LIN {X 0,Y 574.042,Z 450.55,A -85,B 0,C 180,E1 -1993.505,E2 -1993.505} C_VEL
LIN {X 0,Y 573.917,Z 424.53,A -85,B 0,C 180,E1 -1993.836,E2 -1993.836} C_VEL
LIN {X 0,Y 573.507,Z 421.165,A -85,B 0,C 180,E1 -1993.916,E2 -1993.916} C_VEL
LIN {X 0,Y 573.675,Z 396.566,A -85,B 0,C 180,E1 -1996.915,E2 -1996.915} C_VEL
LIN {X 0,Y 573.955,Z 372.952,A -85,B 0,C 180,E1 -1999.849,E2 -1999.849} C_VEL
LIN {X 0,Y 574.301,Z 350.569,A -85,B 0,C 180,E1 -2002.674,E2 -2002.674} C_VEL
LIN {X 0,Y 574.39,Z 334.005,A -85,B 0,C 180,E1 -2004.75,E2 -2004.75} C_VEL
LIN {X 0,Y 573.247,Z 327.79,A -85,B 0,C 180,E1 -2005.605,E2 -2005.605} C_VEL
LIN {X 0,Y 573.252,Z 327.703,A -85,B 0,C 180,E1 -2008.028,E2 -2008.028} C_VEL
LIN {X 0,Y 573.25,Z 327.705,A -85,B 0,C 180,E1 -2010.176,E2 -2010.176} C_VEL
LIN {X 0,Y 573.259,Z 327.704,A -85,B 0,C 180,E1 -2012.645,E2 -2012.645} C_VEL
LIN {X 0,Y 573.21,Z 327.704,A -85,B 0,C 180,E1 -2015.188,E2 -2015.188} C_VEL
LIN {X 0,Y 573.239,Z 327.702,A -85,B 0,C 180,E1 -2017.807,E2 -2017.807} C_VEL
LIN {X 0,Y 573.25,Z 327.704,A -85,B 0,C 180,E1 -2020.525,E2 -2020.525} C_VEL
LIN {X 0,Y 573.245,Z 327.698,A -85,B 0,C 180,E1 -2023.359,E2 -2023.359} C_VEL
LIN {X 0,Y 573.243,Z 327.706,A -85,B 0,C 180,E1 -2026.331,E2 -2026.331} C_VEL
LIN {X 0,Y 573.233,Z 327.703,A -85,B 0,C 180,E1 -2028.542,E2 -2028.542} C_VEL
LIN {X 0,Y 573.248,Z 327.698,A -85,B 0,C 180,E1 -2031.298,E2 -2031.298} C_VEL
LIN {X 0,Y 573.245,Z 327.707,A -85,B 0,C 180,E1 -2034.014,E2 -2034.014} C_VEL
LIN {X 0,Y 573.275,Z 327.697,A -85,B 0,C 180,E1 -2036.517,E2 -2036.517} C_VEL
LIN {X 0,Y 573.234,Z 327.701,A -85,B 0,C 180,E1 -2039.117,E2 -2039.117} C_VEL
LIN {X 0,Y 573.242,Z 327.697,A -85,B 0,C 180,E1 -2041.435,E2 -2041.435} C_VEL
LIN {X 0,Y 573.269,Z 327.702,A -85,B 0,C 180,E1 -2043.81,E2 -2043.81} C_VEL
LIN {X 0,Y 573.238,Z 327.706,A -85,B 0,C 180,E1 -2046.134,E2 -2046.134} C_VEL
LIN {X 0,Y 573.29,Z 327.923,A -85,B 0,C 180,E1 -2046.936,E2 -2046.936} C_VEL
LIN {X 0,Y 574.042,Z 332.774,A -85,B 0,C 180,E1 -2047.694,E2 -2047.694} C_VEL
LIN {X 0,Y 573.791,Z 353.69,A -85,B 0,C 180,E1 -2050.688,E2 -2050.688} C_VEL
LIN {X 0,Y 573.581,Z 371.938,A -85,B 0,C 180,E1 -2053.24,E2 -2053.24} C_VEL
LIN {X 0,Y 573.876,Z 374.016,A -85,B 0,C 180,E1 -2053.322,E2 -2053.322} C_VEL
LIN {X 0,Y 574.602,Z 377.936,A -85,B 0,C 180,E1 -2053.393,E2 -2053.393} C_VEL
LIN {X 0,Y 574.275,Z 508.286,A -85,B 0,C 180,E1 -2055.062,E2 -2055.062} C_VEL
LIN {X 0,Y 574.177,Z 521.251,A -85,B 0,C 180,E1 -2055.339,E2 -2055.339} C_VEL
LIN {X 0,Y 574.097,Z 535.103,A -85,B 0,C 180,E1 -2055.771,E2 -2055.771} C_VEL
LIN {X 0,Y 573.926,Z 548.919,A -85,B 0,C 180,E1 -2056.365,E2 -2056.365} C_VEL
LIN {X 0,Y 573.742,Z 560.44,A -85,B 0,C 180,E1 -2056.991,E2 -2056.991} C_VEL
LIN {X 0,Y 573.599,Z 571.257,A -85,B 0,C 180,E1 -2057.708,E2 -2057.708} C_VEL
LIN {X 0,Y 573.455,Z 581.621,A -85,B 0,C 180,E1 -2058.53,E2 -2058.53} C_VEL
LIN {X 0,Y 573.355,Z 590.92,A -85,B 0,C 180,E1 -2059.404,E2 -2059.404} C_VEL
LIN {X 0,Y 573.256,Z 600.453,A -85,B 0,C 180,E1 -2060.472,E2 -2060.472} C_VEL
LIN {X 0,Y 573.143,Z 609.469,A -85,B 0,C 180,E1 -2061.715,E2 -2061.715} C_VEL
LIN {X 0,Y 573.091,Z 614.888,A -85,B 0,C 180,E1 -2062.601,E2 -2062.601} C_VEL
LIN {X 0,Y 573.022,Z 620.311,A -85,B 0,C 180,E1 -2063.662,E2 -2063.662} C_VEL
LIN {X 0,Y 573,Z 624.764,A -85,B 0,C 180,E1 -2064.721,E2 -2064.721} C_VEL
LIN {X 0,Y 573.029,Z 628.315,A -85,B 0,C 180,E1 -2065.779,E2 -2065.779} C_VEL
LIN {X 0,Y 572.957,Z 631.716,A -85,B 0,C 180,E1 -2067.187,E2 -2067.187} C_VEL
LIN {X 0,Y 572.939,Z 632.942,A -85,B 0,C 180,E1 -2067.89,E2 -2067.89} C_VEL
LIN {X 0,Y 572.936,Z 634.281,A -85,B 0,C 180,E1 -2069.296,E2 -2069.296} C_VEL
LIN {X 0,Y 572.937,Z 634.496,A -85,B 0,C 180,E1 -2069.999,E2 -2069.999} C_VEL
LIN {X 0,Y 572.941,Z 633.863,A -85,B 0,C 180,E1 -2071.405,E2 -2071.405} C_VEL
LIN {X 0,Y 572.954,Z 631.893,A -85,B 0,C 180,E1 -2072.811,E2 -2072.811} C_VEL
LIN {X 0,Y 573.008,Z 630.437,A -85,B 0,C 180,E1 -2073.515,E2 -2073.515} C_VEL
LIN {X 0,Y 572.955,Z 626.342,A -85,B 0,C 180,E1 -2074.925,E2 -2074.925} C_VEL
LIN {X 0,Y 573.044,Z 622.298,A -85,B 0,C 180,E1 -2075.983,E2 -2075.983} C_VEL
LIN {X 0,Y 573.053,Z 617.286,A -85,B 0,C 180,E1 -2077.044,E2 -2077.044} C_VEL
LIN {X 0,Y 573.128,Z 611.185,A -85,B 0,C 180,E1 -2078.106,E2 -2078.106} C_VEL
LIN {X 0,Y 573.219,Z 603.876,A -85,B 0,C 180,E1 -2079.17,E2 -2079.17} C_VEL
LIN {X 0,Y 573.303,Z 595.124,A -85,B 0,C 180,E1 -2080.238,E2 -2080.238} C_VEL
LIN {X 0,Y 573.487,Z 583.882,A -85,B 0,C 180,E1 -2081.365,E2 -2081.365} C_VEL
LIN {X 0,Y 573.585,Z 572.521,A -85,B 0,C 180,E1 -2082.291,E2 -2082.291} C_VEL
LIN {X 0,Y 573.735,Z 561.93,A -85,B 0,C 180,E1 -2083.007,E2 -2083.007} C_VEL
LIN {X 0,Y 573.88,Z 550.7,A -85,B 0,C 180,E1 -2083.634,E2 -2083.634} C_VEL
LIN {X 0,Y 574.013,Z 538.844,A -85,B 0,C 180,E1 -2084.173,E2 -2084.173} C_VEL
LIN {X 0,Y 574.186,Z 523.882,A -85,B 0,C 180,E1 -2084.684,E2 -2084.684} C_VEL
LIN {X 0,Y 574.28,Z 509.711,A -85,B 0,C 180,E1 -2085.004,E2 -2085.004} C_VEL
LIN {X 0,Y 574.423,Z 457.939,A -85,B 0,C 180,E1 -2085.682,E2 -2085.682} C_VEL
LIN {X 0,Y 574.434,Z 376.847,A -85,B 0,C 180,E1 -2086.716,E2 -2086.716} C_VEL
LIN {X 0,Y 573.637,Z 372.312,A -85,B 0,C 180,E1 -2086.819,E2 -2086.819} C_VEL
LIN {X 0,Y 573.702,Z 359.568,A -85,B 0,C 180,E1 -2088.572,E2 -2088.572} C_VEL
LIN {X 0,Y 573.962,Z 340.021,A -85,B 0,C 180,E1 -2091.352,E2 -2091.352} C_VEL
LIN {X 0,Y 574.053,Z 332.1,A -85,B 0,C 180,E1 -2092.493,E2 -2092.493} C_VEL
LIN {X 0,Y 573.275,Z 327.837,A -85,B 0,C 180,E1 -2093.182,E2 -2093.182} C_VEL
LIN {X 0,Y 573.255,Z 327.7,A -85,B 0,C 180,E1 -2095.409,E2 -2095.409} C_VEL
LIN {X 0,Y 573.263,Z 327.705,A -85,B 0,C 180,E1 -2098.031,E2 -2098.031} C_VEL
LIN {X 0,Y 573.243,Z 327.7,A -85,B 0,C 180,E1 -2100.884,E2 -2100.884} C_VEL
LIN {X 0,Y 573.285,Z 327.695,A -85,B 0,C 180,E1 -2103.527,E2 -2103.527} C_VEL
LIN {X 0,Y 573.258,Z 327.705,A -85,B 0,C 180,E1 -2106.047,E2 -2106.047} C_VEL
LIN {X 0,Y 573.246,Z 327.699,A -85,B 0,C 180,E1 -2108.7,E2 -2108.7} C_VEL
LIN {X 0,Y 573.249,Z 327.702,A -85,B 0,C 180,E1 -2111.595,E2 -2111.595} C_VEL
LIN {X 0,Y 573.233,Z 327.7,A -85,B 0,C 180,E1 -2114.332,E2 -2114.332} C_VEL
LIN {X 0,Y 573.254,Z 327.699,A -85,B 0,C 180,E1 -2117.355,E2 -2117.355} C_VEL
LIN {X 0,Y 573.243,Z 327.698,A -85,B 0,C 180,E1 -2120.392,E2 -2120.392} C_VEL
LIN {X 0,Y 573.249,Z 327.695,A -85,B 0,C 180,E1 -2123.077,E2 -2123.077} C_VEL
LIN {X 0,Y 573.265,Z 327.706,A -85,B 0,C 180,E1 -2125.671,E2 -2125.671} C_VEL
LIN {X 0,Y 573.244,Z 327.699,A -85,B 0,C 180,E1 -2128.185,E2 -2128.185} C_VEL
LIN {X 0,Y 573.262,Z 327.69,A -85,B 0,C 180,E1 -2130.634,E2 -2130.634} C_VEL
LIN {X 0,Y 573.264,Z 327.702,A -85,B 0,C 180,E1 -2133.499,E2 -2133.499} C_VEL
LIN {X 0,Y 573.236,Z 327.701,A -85,B 0,C 180,E1 -2136.135,E2 -2136.135} C_VEL
LIN {X 0,Y 573.251,Z 327.697,A -85,B 0,C 180,E1 -2138.706,E2 -2138.706} C_VEL
LIN {X 0,Y 573.233,Z 327.71,A -85,B 0,C 180,E1 -2141.411,E2 -2141.411} C_VEL
LIN {X 0,Y 573.252,Z 327.701,A -85,B 0,C 180,E1 -2143.622,E2 -2143.622} C_VEL
LIN {X 0,Y 573.231,Z 327.7,A -85,B 0,C 180,E1 -2146.529,E2 -2146.529} C_VEL
LIN {X 0,Y 573.272,Z 327.7,A -85,B 0,C 180,E1 -2149.403,E2 -2149.403} C_VEL
LIN {X 0,Y 573.282,Z 327.693,A -85,B 0,C 180,E1 -2152.25,E2 -2152.25} C_VEL
LIN {X 0,Y 573.307,Z 327.7,A -85,B 0,C 180,E1 -2155.077,E2 -2155.077} C_VEL
LIN {X 0,Y 573.301,Z 327.691,A -85,B 0,C 180,E1 -2157.892,E2 -2157.892} C_VEL
LIN {X 0,Y 573.333,Z 327.693,A -85,B 0,C 180,E1 -2160.702,E2 -2160.702} C_VEL
LIN {X 0,Y 573.237,Z 327.7,A -85,B 0,C 180,E1 -2163.514,E2 -2163.514} C_VEL
LIN {X 0,Y 573.288,Z 327.694,A -85,B 0,C 180,E1 -2165.628,E2 -2165.628} C_VEL
LIN {X 0,Y 573.299,Z 327.695,A -85,B 0,C 180,E1 -2168.459,E2 -2168.459} C_VEL
LIN {X 0,Y 573.288,Z 327.695,A -85,B 0,C 180,E1 -2171.312,E2 -2171.312} C_VEL
LIN {X 0,Y 573.271,Z 327.699,A -85,B 0,C 180,E1 -2174.425,E2 -2174.425} C_VEL
LIN {X 0,Y 573.252,Z 327.701,A -85,B 0,C 180,E1 -2177.112,E2 -2177.112} C_VEL
LIN {X 0,Y 573.25,Z 327.699,A -85,B 0,C 180,E1 -2180.077,E2 -2180.077} C_VEL
LIN {X 0,Y 573.262,Z 327.698,A -85,B 0,C 180,E1 -2183.154,E2 -2183.154} C_VEL
LIN {X 0,Y 573.28,Z 327.698,A -85,B 0,C 180,E1 -2186.189,E2 -2186.189} C_VEL
LIN {X 0,Y 573.235,Z 327.701,A -85,B 0,C 180,E1 -2188.565,E2 -2188.565} C_VEL
LIN {X 0,Y 573.229,Z 327.701,A -85,B 0,C 180,E1 -2190.993,E2 -2190.993} C_VEL
LIN {X 0,Y 573.279,Z 327.695,A -85,B 0,C 180,E1 -2193.529,E2 -2193.529} C_VEL
LIN {X 0,Y 573.252,Z 327.702,A -85,B 0,C 180,E1 -2196.049,E2 -2196.049} C_VEL
LIN {X 0,Y 573.241,Z 327.701,A -85,B 0,C 180,E1 -2198.702,E2 -2198.702} C_VEL
LIN {X 0,Y 573.258,Z 327.699,A -85,B 0,C 180,E1 -2201.598,E2 -2201.598} C_VEL
LIN {X 0,Y 573.232,Z 327.704,A -85,B 0,C 180,E1 -2204.334,E2 -2204.334} C_VEL
LIN {X 0,Y 573.237,Z 327.7,A -85,B 0,C 180,E1 -2207.359,E2 -2207.359} C_VEL
LIN {X 0,Y 573.245,Z 327.703,A -85,B 0,C 180,E1 -2210.394,E2 -2210.394} C_VEL
LIN {X 0,Y 573.252,Z 327.698,A -85,B 0,C 180,E1 -2213.079,E2 -2213.079} C_VEL
LIN {X 0,Y 573.272,Z 327.701,A -85,B 0,C 180,E1 -2215.673,E2 -2215.673} C_VEL
LIN {X 0,Y 573.247,Z 327.705,A -85,B 0,C 180,E1 -2218.186,E2 -2218.186} C_VEL
LIN {X 0,Y 573.268,Z 327.691,A -85,B 0,C 180,E1 -2220.636,E2 -2220.636} C_VEL
LIN {X 0,Y 573.267,Z 327.702,A -85,B 0,C 180,E1 -2223.502,E2 -2223.502} C_VEL
LIN {X 0,Y 573.232,Z 327.707,A -85,B 0,C 180,E1 -2226.136,E2 -2226.136} C_VEL
LIN {X 0,Y 573.26,Z 327.868,A -85,B 0,C 180,E1 -2226.875,E2 -2226.875} C_VEL
LIN {X 0,Y 574.085,Z 333.097,A -85,B 0,C 180,E1 -2227.698,E2 -2227.698} C_VEL
LIN {X 0,Y 573.784,Z 354.019,A -85,B 0,C 180,E1 -2230.689,E2 -2230.689} C_VEL
LIN {X 0,Y 573.608,Z 372.016,A -85,B 0,C 180,E1 -2233.203,E2 -2233.203} C_VEL
LIN {X 0,Y 574.046,Z 374.736,A -85,B 0,C 180,E1 -2233.291,E2 -2233.291} C_VEL
LIN {X 0,Y 574.6,Z 379.508,A -85,B 0,C 180,E1 -2233.368,E2 -2233.368} C_VEL
LIN {X 0,Y 574.303,Z 508.7,A -85,B 0,C 180,E1 -2235.019,E2 -2235.019} C_VEL
LIN {X 0,Y 574.186,Z 523.423,A -85,B 0,C 180,E1 -2235.349,E2 -2235.349} C_VEL
LIN {X 0,Y 574.02,Z 537.729,A -85,B 0,C 180,E1 -2235.827,E2 -2235.827} C_VEL
LIN {X 0,Y 573.889,Z 551.665,A -85,B 0,C 180,E1 -2236.456,E2 -2236.456} C_VEL
LIN {X 0,Y 573.717,Z 564.118,A -85,B 0,C 180,E1 -2237.173,E2 -2237.173} C_VEL
LIN {X 0,Y 573.532,Z 576.655,A -85,B 0,C 180,E1 -2238.067,E2 -2238.067} C_VEL
LIN {X 0,Y 573.435,Z 588.186,A -85,B 0,C 180,E1 -2239.084,E2 -2239.084} C_VEL
LIN {X 0,Y 573.239,Z 597.86,A -85,B 0,C 180,E1 -2240.118,E2 -2240.118} C_VEL
LIN {X 0,Y 573.201,Z 606.179,A -85,B 0,C 180,E1 -2241.185,E2 -2241.185} C_VEL
LIN {X 0,Y 573.109,Z 614.133,A -85,B 0,C 180,E1 -2242.426,E2 -2242.426} C_VEL
LIN {X 0,Y 573.02,Z 620.531,A -85,B 0,C 180,E1 -2243.664,E2 -2243.664} C_VEL
LIN {X 0,Y 573.001,Z 624.964,A -85,B 0,C 180,E1 -2244.723,E2 -2244.723} C_VEL
LIN {X 0,Y 573.028,Z 628.447,A -85,B 0,C 180,E1 -2245.781,E2 -2245.781} C_VEL
LIN {X 0,Y 572.956,Z 631.835,A -85,B 0,C 180,E1 -2247.189,E2 -2247.189} C_VEL
LIN {X 0,Y 572.941,Z 633.834,A -85,B 0,C 180,E1 -2248.595,E2 -2248.595} C_VEL
LIN {X 0,Y 572.937,Z 634.5,A -85,B 0,C 180,E1 -2250.001,E2 -2250.001} C_VEL
LIN {X 0,Y 572.941,Z 633.832,A -85,B 0,C 180,E1 -2251.407,E2 -2251.407} C_VEL
LIN {X 0,Y 572.956,Z 631.83,A -85,B 0,C 180,E1 -2252.813,E2 -2252.813} C_VEL
LIN {X 0,Y 573.028,Z 628.44,A -85,B 0,C 180,E1 -2254.221,E2 -2254.221} C_VEL
LIN {X 0,Y 573.059,Z 623.565,A -85,B 0,C 180,E1 -2255.631,E2 -2255.631} C_VEL
LIN {X 0,Y 573.059,Z 618.85,A -85,B 0,C 180,E1 -2256.693,E2 -2256.693} C_VEL
LIN {X 0,Y 573.126,Z 612.031,A -85,B 0,C 180,E1 -2257.93,E2 -2257.93} C_VEL
LIN {X 0,Y 573.226,Z 603.552,A -85,B 0,C 180,E1 -2259.172,E2 -2259.172} C_VEL
LIN {X 0,Y 573.305,Z 594.7,A -85,B 0,C 180,E1 -2260.24,E2 -2260.24} C_VEL
LIN {X 0,Y 573.464,Z 583.982,A -85,B 0,C 180,E1 -2261.309,E2 -2261.309} C_VEL
LIN {X 0,Y 573.618,Z 573.131,A -85,B 0,C 180,E1 -2262.202,E2 -2262.202} C_VEL
LIN {X 0,Y 573.741,Z 561.243,A -85,B 0,C 180,E1 -2263.009,E2 -2263.009} C_VEL
LIN {X 0,Y 573.947,Z 548.081,A -85,B 0,C 180,E1 -2263.725,E2 -2263.725} C_VEL
LIN {X 0,Y 574.085,Z 534.8,A -85,B 0,C 180,E1 -2264.285,E2 -2264.285} C_VEL
LIN {X 0,Y 574.208,Z 520.713,A -85,B 0,C 180,E1 -2264.722,E2 -2264.722} C_VEL
LIN {X 0,Y 574.315,Z 507.08,A -85,B 0,C 180,E1 -2265.005,E2 -2265.005} C_VEL
LIN {X 0,Y 574.467,Z 376.987,A -85,B 0,C 180,E1 -2266.668,E2 -2266.668} C_VEL
LIN {X 0,Y 573.617,Z 372.383,A -85,B 0,C 180,E1 -2266.77,E2 -2266.77} C_VEL
LIN {X 0,Y 573.621,Z 368.522,A -85,B 0,C 180,E1 -2267.266,E2 -2267.266} C_VEL
LIN {X 0,Y 573.892,Z 346.16,A -85,B 0,C 180,E1 -2270.428,E2 -2270.428} C_VEL
LIN {X 0,Y 574.034,Z 331.776,A -85,B 0,C 180,E1 -2272.496,E2 -2272.496} C_VEL
LIN {X 0,Y 573.262,Z 327.809,A -85,B 0,C 180,E1 -2273.15,E2 -2273.15} C_VEL
LIN {X 0,Y 573.258,Z 327.699,A -85,B 0,C 180,E1 -2275.411,E2 -2275.411} C_VEL
LIN {X 0,Y 573.269,Z 327.703,A -85,B 0,C 180,E1 -2278.032,E2 -2278.032} C_VEL
LIN {X 0,Y 573.234,Z 327.701,A -85,B 0,C 180,E1 -2280.883,E2 -2280.883} C_VEL
LIN {X 0,Y 573.267,Z 327.698,A -85,B 0,C 180,E1 -2283.524,E2 -2283.524} C_VEL
LIN {X 0,Y 573.266,Z 327.705,A -85,B 0,C 180,E1 -2286.048,E2 -2286.048} C_VEL
LIN {X 0,Y 573.247,Z 327.7,A -85,B 0,C 180,E1 -2288.702,E2 -2288.702} C_VEL
LIN {X 0,Y 573.234,Z 327.705,A -85,B 0,C 180,E1 -2291.593,E2 -2291.593} C_VEL
LIN {X 0,Y 573.233,Z 327.704,A -85,B 0,C 180,E1 -2294.334,E2 -2294.334} C_VEL
LIN {X 0,Y 573.245,Z 327.702,A -85,B 0,C 180,E1 -2297.359,E2 -2297.359} C_VEL
LIN {X 0,Y 573.243,Z 327.701,A -85,B 0,C 180,E1 -2300.393,E2 -2300.393} C_VEL
LIN {X 0,Y 573.256,Z 327.699,A -85,B 0,C 180,E1 -2303.078,E2 -2303.078} C_VEL
LIN {X 0,Y 573.27,Z 327.706,A -85,B 0,C 180,E1 -2305.671,E2 -2305.671} C_VEL
LIN {X 0,Y 573.245,Z 327.702,A -85,B 0,C 180,E1 -2308.185,E2 -2308.185} C_VEL
LIN {X 0,Y 573.268,Z 327.697,A -85,B 0,C 180,E1 -2310.634,E2 -2310.634} C_VEL
LIN {X 0,Y 573.255,Z 327.702,A -85,B 0,C 180,E1 -2313.024,E2 -2313.024} C_VEL
LIN {X 0,Y 573.3,Z 327.912,A -85,B 0,C 180,E1 -2314.607,E2 -2314.607} C_VEL
LIN {X 0,Y 574.331,Z 334.315,A -85,B 0,C 180,E1 -2315.414,E2 -2315.414} C_VEL
LIN {X 0,Y 574.197,Z 352.833,A -85,B 0,C 180,E1 -2317.702,E2 -2317.702} C_VEL
LIN {X 0,Y 573.943,Z 373.525,A -85,B 0,C 180,E1 -2320.313,E2 -2320.313} C_VEL
LIN {X 0,Y 573.687,Z 397.322,A -85,B 0,C 180,E1 -2323.268,E2 -2323.268} C_VEL
LIN {X 0,Y 573.472,Z 420.909,A -85,B 0,C 180,E1 -2326.151,E2 -2326.151} C_VEL
LIN {X 0,Y 573.649,Z 422.658,A -85,B 0,C 180,E1 -2326.223,E2 -2326.223} C_VEL
LIN {X 0,Y 574.082,Z 429.808,A -85,B 0,C 180,E1 -2326.324,E2 -2326.324} C_VEL
LIN {X 0,Y 573.866,Z 530.384,A -85,B 0,C 180,E1 -2327.602,E2 -2327.602} C_VEL
LIN {X 0,Y 573.813,Z 543.76,A -85,B 0,C 180,E1 -2327.915,E2 -2327.915} C_VEL
LIN {X 0,Y 573.717,Z 555.894,A -85,B 0,C 180,E1 -2328.339,E2 -2328.339} C_VEL
LIN {X 0,Y 573.623,Z 567.331,A -85,B 0,C 180,E1 -2328.877,E2 -2328.877} C_VEL
LIN {X 0,Y 573.432,Z 579.073,A -85,B 0,C 180,E1 -2329.585,E2 -2329.585} C_VEL
LIN {X 0,Y 573.329,Z 589.575,A -85,B 0,C 180,E1 -2330.386,E2 -2330.386} C_VEL
LIN {X 0,Y 573.244,Z 599.888,A -85,B 0,C 180,E1 -2331.362,E2 -2331.362} C_VEL
LIN {X 0,Y 573.143,Z 608.856,A -85,B 0,C 180,E1 -2332.425,E2 -2332.425} C_VEL
LIN {X 0,Y 573.104,Z 615.339,A -85,B 0,C 180,E1 -2333.37,E2 -2333.37} C_VEL
LIN {X 0,Y 573.071,Z 620.956,A -85,B 0,C 180,E1 -2334.37,E2 -2334.37} C_VEL
LIN {X 0,Y 573.028,Z 625.694,A -85,B 0,C 180,E1 -2335.428,E2 -2335.428} C_VEL
LIN {X 0,Y 573.023,Z 629.324,A -85,B 0,C 180,E1 -2336.484,E2 -2336.484} C_VEL
LIN {X 0,Y 572.959,Z 631.194,A -85,B 0,C 180,E1 -2337.188,E2 -2337.188} C_VEL
LIN {X 0,Y 572.938,Z 632.629,A -85,B 0,C 180,E1 -2337.891,E2 -2337.891} C_VEL
LIN {X 0,Y 572.941,Z 634.254,A -85,B 0,C 180,E1 -2339.297,E2 -2339.297} C_VEL
LIN {X 0,Y 572.938,Z 634.496,A -85,B 0,C 180,E1 -2340,E2 -2340} C_VEL
LIN {X 0,Y 572.941,Z 634.314,A -85,B 0,C 180,E1 -2340.703,E2 -2340.703} C_VEL
LIN {X 0,Y 572.937,Z 632.77,A -85,B 0,C 180,E1 -2342.109,E2 -2342.109} C_VEL
LIN {X 0,Y 572.96,Z 631.411,A -85,B 0,C 180,E1 -2342.812,E2 -2342.812} C_VEL
LIN {X 0,Y 573.015,Z 628.538,A -85,B 0,C 180,E1 -2343.868,E2 -2343.868} C_VEL
LIN {X 0,Y 572.963,Z 624.639,A -85,B 0,C 180,E1 -2344.926,E2 -2344.926} C_VEL
LIN {X 0,Y 573.073,Z 619.607,A -85,B 0,C 180,E1 -2345.984,E2 -2345.984} C_VEL
LIN {X 0,Y 573.084,Z 613.265,A -85,B 0,C 180,E1 -2347.044,E2 -2347.044} C_VEL
LIN {X 0,Y 573.175,Z 605.366,A -85,B 0,C 180,E1 -2348.106,E2 -2348.106} C_VEL
LIN {X 0,Y 573.254,Z 597.295,A -85,B 0,C 180,E1 -2348.993,E2 -2348.993} C_VEL
LIN {X 0,Y 573.338,Z 587.451,A -85,B 0,C 180,E1 -2349.882,E2 -2349.882} C_VEL
LIN {X 0,Y 573.51,Z 576.394,A -85,B 0,C 180,E1 -2350.681,E2 -2350.681} C_VEL
LIN {X 0,Y 573.614,Z 564.162,A -85,B 0,C 180,E1 -2351.378,E2 -2351.378} C_VEL
LIN {X 0,Y 573.738,Z 551.494,A -85,B 0,C 180,E1 -2351.921,E2 -2351.921} C_VEL
LIN {X 0,Y 573.837,Z 538.826,A -85,B 0,C 180,E1 -2352.309,E2 -2352.309} C_VEL
LIN {X 0,Y 573.948,Z 526.185,A -85,B 0,C 180,E1 -2352.553,E2 -2352.553} C_VEL
LIN {X 0,Y 574.042,Z 450.55,A -85,B 0,C 180,E1 -2353.505,E2 -2353.505} C_VEL
LIN {X 0,Y 573.357,Z 446.676,A -85,B 0,C 180,E1 -2353.57,E2 -2353.57} C_VEL
LIN {X 0,Y 567.856,Z 434.691,A -85,B 0,C 180,E1 -2353.857,E2 -2353.857} C_VEL
LIN {X 0,Y 567.19,Z 430.818,A -85,B 0,C 180,E1 -2353.923,E2 -2353.923} C_VEL
LIN {X 0,Y 566.942,Z 424.77,A -85,B 0,C 180,E1 -2354.006,E2 -2354.006} C_VEL
LIN {X 0,Y 566.535,Z 421.158,A -85,B 0,C 180,E1 -2354.091,E2 -2354.091} C_VEL
LIN {X 0,Y 566.721,Z 396.453,A -85,B 0,C 180,E1 -2357.143,E2 -2357.143} C_VEL
LIN {X 0,Y 567.068,Z 372.969,A -85,B 0,C 180,E1 -2360.097,E2 -2360.097} C_VEL
LIN {X 0,Y 567.396,Z 351.815,A -85,B 0,C 180,E1 -2362.773,E2 -2362.773} C_VEL
LIN {X 0,Y 567.44,Z 334.835,A -85,B 0,C 180,E1 -2364.905,E2 -2364.905} C_VEL
LIN {X 0,Y 566.218,Z 328.668,A -85,B 0,C 180,E1 -2365.774,E2 -2365.774} C_VEL
LIN {X 0,Y 566.208,Z 328.582,A -85,B 0,C 180,E1 -2368.202,E2 -2368.202} C_VEL
LIN {X 0,Y 566.195,Z 328.579,A -85,B 0,C 180,E1 -2371.076,E2 -2371.076} C_VEL
LIN {X 0,Y 566.217,Z 328.576,A -85,B 0,C 180,E1 -2373.734,E2 -2373.734} C_VEL
LIN {X 0,Y 566.204,Z 328.582,A -85,B 0,C 180,E1 -2376.57,E2 -2376.57} C_VEL
LIN {X 0,Y 566.219,Z 328.576,A -85,B 0,C 180,E1 -2379.685,E2 -2379.685} C_VEL
LIN {X 0,Y 566.207,Z 328.575,A -85,B 0,C 180,E1 -2382.917,E2 -2382.917} C_VEL
LIN {X 0,Y 566.199,Z 328.581,A -85,B 0,C 180,E1 -2386.049,E2 -2386.049} C_VEL
LIN {X 0,Y 566.209,Z 328.575,A -85,B 0,C 180,E1 -2389.214,E2 -2389.214} C_VEL
LIN {X 0,Y 566.191,Z 328.58,A -85,B 0,C 180,E1 -2391.637,E2 -2391.637} C_VEL
LIN {X 0,Y 566.199,Z 328.582,A -85,B 0,C 180,E1 -2394.31,E2 -2394.31} C_VEL
LIN {X 0,Y 566.225,Z 328.573,A -85,B 0,C 180,E1 -2396.897,E2 -2396.897} C_VEL
LIN {X 0,Y 566.187,Z 328.581,A -85,B 0,C 180,E1 -2399.407,E2 -2399.407} C_VEL
LIN {X 0,Y 566.217,Z 328.578,A -85,B 0,C 180,E1 -2401.857,E2 -2401.857} C_VEL
LIN {X 0,Y 566.219,Z 328.576,A -85,B 0,C 180,E1 -2404.251,E2 -2404.251} C_VEL
LIN {X 0,Y 566.216,Z 328.717,A -85,B 0,C 180,E1 -2406.74,E2 -2406.74} C_VEL
LIN {X 0,Y 567.137,Z 334.085,A -85,B 0,C 180,E1 -2407.6,E2 -2407.6} C_VEL
LIN {X 0,Y 566.875,Z 353.694,A -85,B 0,C 180,E1 -2410.442,E2 -2410.442} C_VEL
LIN {X 0,Y 566.655,Z 372.243,A -85,B 0,C 180,E1 -2413.053,E2 -2413.053} C_VEL
LIN {X 0,Y 567.811,Z 379.084,A -85,B 0,C 180,E1 -2413.203,E2 -2413.203} C_VEL
LIN {X 0,Y 567.428,Z 508.264,A -85,B 0,C 180,E1 -2414.877,E2 -2414.877} C_VEL
LIN {X 0,Y 567.324,Z 520.71,A -85,B 0,C 180,E1 -2415.144,E2 -2415.144} C_VEL
LIN {X 0,Y 567.249,Z 533.726,A -85,B 0,C 180,E1 -2415.546,E2 -2415.546} C_VEL
LIN {X 0,Y 567.061,Z 547.147,A -85,B 0,C 180,E1 -2416.105,E2 -2416.105} C_VEL
LIN {X 0,Y 566.813,Z 558.973,A -85,B 0,C 180,E1 -2416.738,E2 -2416.738} C_VEL
LIN {X 0,Y 566.651,Z 570.013,A -85,B 0,C 180,E1 -2417.464,E2 -2417.464} C_VEL
LIN {X 0,Y 566.502,Z 580.35,A -85,B 0,C 180,E1 -2418.278,E2 -2418.278} C_VEL
LIN {X 0,Y 566.4,Z 589.455,A -85,B 0,C 180,E1 -2419.125,E2 -2419.125} C_VEL
LIN {X 0,Y 566.199,Z 598.972,A -85,B 0,C 180,E1 -2420.172,E2 -2420.172} C_VEL
LIN {X 0,Y 566.091,Z 608.334,A -85,B 0,C 180,E1 -2421.431,E2 -2421.431} C_VEL
LIN {X 0,Y 566.017,Z 614.887,A -85,B 0,C 180,E1 -2422.508,E2 -2422.508} C_VEL
LIN {X 0,Y 565.946,Z 620.313,A -85,B 0,C 180,E1 -2423.582,E2 -2423.582} C_VEL
LIN {X 0,Y 565.928,Z 624.76,A -85,B 0,C 180,E1 -2424.655,E2 -2424.655} C_VEL
LIN {X 0,Y 565.957,Z 628.317,A -85,B 0,C 180,E1 -2425.726,E2 -2425.726} C_VEL
LIN {X 0,Y 565.875,Z 631.71,A -85,B 0,C 180,E1 -2427.152,E2 -2427.152} C_VEL
LIN {X 0,Y 565.84,Z 632.944,A -85,B 0,C 180,E1 -2427.864,E2 -2427.864} C_VEL
LIN {X 0,Y 565.836,Z 634.274,A -85,B 0,C 180,E1 -2429.287,E2 -2429.287} C_VEL
LIN {X 0,Y 565.838,Z 634.496,A -85,B 0,C 180,E1 -2429.999,E2 -2429.999} C_VEL
LIN {X 0,Y 565.841,Z 633.859,A -85,B 0,C 180,E1 -2431.423,E2 -2431.423} C_VEL
LIN {X 0,Y 565.873,Z 631.884,A -85,B 0,C 180,E1 -2432.847,E2 -2432.847} C_VEL
LIN {X 0,Y 565.914,Z 630.436,A -85,B 0,C 180,E1 -2433.559,E2 -2433.559} C_VEL
LIN {X 0,Y 565.929,Z 627.533,A -85,B 0,C 180,E1 -2434.629,E2 -2434.629} C_VEL
LIN {X 0,Y 565.961,Z 622.288,A -85,B 0,C 180,E1 -2436.058,E2 -2436.058} C_VEL
LIN {X 0,Y 565.98,Z 617.274,A -85,B 0,C 180,E1 -2437.132,E2 -2437.132} C_VEL
LIN {X 0,Y 566.055,Z 611.174,A -85,B 0,C 180,E1 -2438.208,E2 -2438.208} C_VEL
LIN {X 0,Y 566.171,Z 603.863,A -85,B 0,C 180,E1 -2439.286,E2 -2439.286} C_VEL
LIN {X 0,Y 566.282,Z 595.108,A -85,B 0,C 180,E1 -2440.366,E2 -2440.366} C_VEL
LIN {X 0,Y 566.467,Z 583.527,A -85,B 0,C 180,E1 -2441.539,E2 -2441.539} C_VEL
LIN {X 0,Y 566.624,Z 572.499,A -85,B 0,C 180,E1 -2442.444,E2 -2442.444} C_VEL
LIN {X 0,Y 566.768,Z 561.905,A -85,B 0,C 180,E1 -2443.17,E2 -2443.17} C_VEL
LIN {X 0,Y 566.952,Z 550.676,A -85,B 0,C 180,E1 -2443.804,E2 -2443.804} C_VEL
LIN {X 0,Y 567.124,Z 538.807,A -85,B 0,C 180,E1 -2444.349,E2 -2444.349} C_VEL
LIN {X 0,Y 567.306,Z 523.897,A -85,B 0,C 180,E1 -2444.865,E2 -2444.865} C_VEL
LIN {X 0,Y 567.429,Z 509.62,A -85,B 0,C 180,E1 -2445.19,E2 -2445.19} C_VEL
LIN {X 0,Y 567.603,Z 465.05,A -85,B 0,C 180,E1 -2445.783,E2 -2445.783} C_VEL
LIN {X 0,Y 567.734,Z 378.263,A -85,B 0,C 180,E1 -2446.9,E2 -2446.9} C_VEL
LIN {X 0,Y 566.678,Z 372.25,A -85,B 0,C 180,E1 -2447.036,E2 -2447.036} C_VEL
LIN {X 0,Y 566.879,Z 353.156,A -85,B 0,C 180,E1 -2449.725,E2 -2449.725} C_VEL
LIN {X 0,Y 567.139,Z 333.403,A -85,B 0,C 180,E1 -2452.59,E2 -2452.59} C_VEL
LIN {X 0,Y 566.214,Z 328.711,A -85,B 0,C 180,E1 -2453.354,E2 -2453.354} C_VEL
LIN {X 0,Y 566.224,Z 328.575,A -85,B 0,C 180,E1 -2455.747,E2 -2455.747} C_VEL
LIN {X 0,Y 566.205,Z 328.58,A -85,B 0,C 180,E1 -2458.202,E2 -2458.202} C_VEL
LIN {X 0,Y 566.193,Z 328.581,A -85,B 0,C 180,E1 -2460.591,E2 -2460.591} C_VEL
LIN {X 0,Y 566.226,Z 328.572,A -85,B 0,C 180,E1 -2463.1,E2 -2463.1} C_VEL
LIN {X 0,Y 566.21,Z 328.579,A -85,B 0,C 180,E1 -2465.687,E2 -2465.687} C_VEL
LIN {X 0,Y 566.213,Z 328.576,A -85,B 0,C 180,E1 -2468.558,E2 -2468.558} C_VEL
LIN {X 0,Y 566.207,Z 328.575,A -85,B 0,C 180,E1 -2471.135,E2 -2471.135} C_VEL
LIN {X 0,Y 566.194,Z 328.581,A -85,B 0,C 180,E1 -2474.034,E2 -2474.034} C_VEL
LIN {X 0,Y 566.208,Z 328.575,A -85,B 0,C 180,E1 -2477.08,E2 -2477.08} C_VEL
LIN {X 0,Y 566.22,Z 328.581,A -85,B 0,C 180,E1 -2479.802,E2 -2479.802} C_VEL
LIN {X 0,Y 566.192,Z 328.572,A -85,B 0,C 180,E1 -2482.598,E2 -2482.598} C_VEL
LIN {X 0,Y 566.212,Z 328.576,A -85,B 0,C 180,E1 -2485.182,E2 -2485.182} C_VEL
LIN {X 0,Y 566.229,Z 328.579,A -85,B 0,C 180,E1 -2487.743,E2 -2487.743} C_VEL
LIN {X 0,Y 566.22,Z 328.567,A -85,B 0,C 180,E1 -2490.322,E2 -2490.322} C_VEL
LIN {X 0,Y 566.228,Z 328.575,A -85,B 0,C 180,E1 -2493.334,E2 -2493.334} C_VEL
LIN {X 0,Y 566.196,Z 328.581,A -85,B 0,C 180,E1 -2495.819,E2 -2495.819} C_VEL
LIN {X 0,Y 566.209,Z 328.575,A -85,B 0,C 180,E1 -2498.902,E2 -2498.902} C_VEL
LIN {X 0,Y 566.206,Z 328.581,A -85,B 0,C 180,E1 -2501.172,E2 -2501.172} C_VEL
LIN {X 0,Y 566.215,Z 328.58,A -85,B 0,C 180,E1 -2503.412,E2 -2503.412} C_VEL
LIN {X 0,Y 566.193,Z 328.576,A -85,B 0,C 180,E1 -2506.359,E2 -2506.359} C_VEL
LIN {X 0,Y 566.265,Z 328.569,A -85,B 0,C 180,E1 -2508.654,E2 -2508.654} C_VEL
LIN {X 0,Y 566.241,Z 328.576,A -85,B 0,C 180,E1 -2511.434,E2 -2511.434} C_VEL
LIN {X 0,Y 566.255,Z 328.569,A -85,B 0,C 180,E1 -2514.302,E2 -2514.302} C_VEL
LIN {X 0,Y 566.272,Z 328.566,A -85,B 0,C 180,E1 -2517.866,E2 -2517.866} C_VEL
LIN {X 0,Y 566.302,Z 328.569,A -85,B 0,C 180,E1 -2520.711,E2 -2520.711} C_VEL
LIN {X 0,Y 566.273,Z 328.574,A -85,B 0,C 180,E1 -2522.846,E2 -2522.846} C_VEL
LIN {X 0,Y 566.255,Z 328.57,A -85,B 0,C 180,E1 -2525.698,E2 -2525.698} C_VEL
LIN {X 0,Y 566.241,Z 328.575,A -85,B 0,C 180,E1 -2528.565,E2 -2528.565} C_VEL
LIN {X 0,Y 566.241,Z 328.572,A -85,B 0,C 180,E1 -2531.454,E2 -2531.454} C_VEL
LIN {X 0,Y 566.224,Z 328.578,A -85,B 0,C 180,E1 -2534.507,E2 -2534.507} C_VEL
LIN {X 0,Y 566.197,Z 328.577,A -85,B 0,C 180,E1 -2537.332,E2 -2537.332} C_VEL
LIN {X 0,Y 566.212,Z 328.579,A -85,B 0,C 180,E1 -2540.337,E2 -2540.337} C_VEL
LIN {X 0,Y 566.221,Z 328.574,A -85,B 0,C 180,E1 -2543.402,E2 -2543.402} C_VEL
LIN {X 0,Y 566.216,Z 328.574,A -85,B 0,C 180,E1 -2545.749,E2 -2545.749} C_VEL
LIN {X 0,Y 566.199,Z 328.577,A -85,B 0,C 180,E1 -2548.204,E2 -2548.204} C_VEL
LIN {X 0,Y 566.191,Z 328.577,A -85,B 0,C 180,E1 -2551.079,E2 -2551.079} C_VEL
LIN {X 0,Y 566.22,Z 328.575,A -85,B 0,C 180,E1 -2553.738,E2 -2553.738} C_VEL
LIN {X 0,Y 566.208,Z 328.576,A -85,B 0,C 180,E1 -2556.569,E2 -2556.569} C_VEL
LIN {X 0,Y 566.206,Z 328.575,A -85,B 0,C 180,E1 -2559.687,E2 -2559.687} C_VEL
LIN {X 0,Y 566.222,Z 328.581,A -85,B 0,C 180,E1 -2562.087,E2 -2562.087} C_VEL
LIN {X 0,Y 566.167,Z 328.577,A -85,B 0,C 180,E1 -2565.037,E2 -2565.037} C_VEL
LIN {X 0,Y 566.213,Z 328.583,A -85,B 0,C 180,E1 -2568.137,E2 -2568.137} C_VEL
LIN {X 0,Y 566.219,Z 328.574,A -85,B 0,C 180,E1 -2570.728,E2 -2570.728} C_VEL
LIN {X 0,Y 566.214,Z 328.581,A -85,B 0,C 180,E1 -2573.784,E2 -2573.784} C_VEL
LIN {X 0,Y 566.226,Z 328.577,A -85,B 0,C 180,E1 -2576.264,E2 -2576.264} C_VEL
LIN {X 0,Y 566.2,Z 328.577,A -85,B 0,C 180,E1 -2578.922,E2 -2578.922} C_VEL
LIN {X 0,Y 566.194,Z 328.572,A -85,B 0,C 180,E1 -2581.048,E2 -2581.048} C_VEL
LIN {X 0,Y 566.243,Z 328.577,A -85,B 0,C 180,E1 -2583.461,E2 -2583.461} C_VEL
LIN {X 0,Y 566.198,Z 328.584,A -85,B 0,C 180,E1 -2585.82,E2 -2585.82} C_VEL
LIN {X 0,Y 566.22,Z 328.761,A -85,B 0,C 180,E1 -2586.708,E2 -2586.708} C_VEL
LIN {X 0,Y 567.176,Z 334.405,A -85,B 0,C 180,E1 -2587.604,E2 -2587.604} C_VEL
LIN {X 0,Y 566.843,Z 354.796,A -85,B 0,C 180,E1 -2590.555,E2 -2590.555} C_VEL
LIN {X 0,Y 566.645,Z 372.178,A -85,B 0,C 180,E1 -2593.003,E2 -2593.003} C_VEL
LIN {X 0,Y 567.613,Z 377.668,A -85,B 0,C 180,E1 -2593.134,E2 -2593.134} C_VEL
LIN {X 0,Y 567.564,Z 470.5,A -85,B 0,C 180,E1 -2594.331,E2 -2594.331} C_VEL
LIN {X 0,Y 567.448,Z 509.936,A -85,B 0,C 180,E1 -2594.857,E2 -2594.857} C_VEL
LIN {X 0,Y 567.279,Z 524.467,A -85,B 0,C 180,E1 -2595.198,E2 -2595.198} C_VEL
LIN {X 0,Y 567.128,Z 538.857,A -85,B 0,C 180,E1 -2595.697,E2 -2595.697} C_VEL
LIN {X 0,Y 566.971,Z 551.664,A -85,B 0,C 180,E1 -2596.288,E2 -2596.288} C_VEL
LIN {X 0,Y 566.771,Z 564.12,A -85,B 0,C 180,E1 -2597.013,E2 -2597.013} C_VEL
LIN {X 0,Y 566.575,Z 576.656,A -85,B 0,C 180,E1 -2597.918,E2 -2597.918} C_VEL
LIN {X 0,Y 566.444,Z 587.329,A -85,B 0,C 180,E1 -2598.862,E2 -2598.862} C_VEL
LIN {X 0,Y 566.205,Z 597.86,A -85,B 0,C 180,E1 -2599.994,E2 -2599.994} C_VEL
LIN {X 0,Y 566.132,Z 606.18,A -85,B 0,C 180,E1 -2601.074,E2 -2601.074} C_VEL
LIN {X 0,Y 566.045,Z 614.133,A -85,B 0,C 180,E1 -2602.331,E2 -2602.331} C_VEL
LIN {X 0,Y 565.943,Z 620.531,A -85,B 0,C 180,E1 -2603.584,E2 -2603.584} C_VEL
LIN {X 0,Y 565.928,Z 624.964,A -85,B 0,C 180,E1 -2604.657,E2 -2604.657} C_VEL
LIN {X 0,Y 565.956,Z 628.448,A -85,B 0,C 180,E1 -2605.728,E2 -2605.728} C_VEL
LIN {X 0,Y 565.874,Z 631.836,A -85,B 0,C 180,E1 -2607.153,E2 -2607.153} C_VEL
LIN {X 0,Y 565.84,Z 633.835,A -85,B 0,C 180,E1 -2608.577,E2 -2608.577} C_VEL
LIN {X 0,Y 565.837,Z 634.5,A -85,B 0,C 180,E1 -2610.001,E2 -2610.001} C_VEL
LIN {X 0,Y 565.84,Z 633.832,A -85,B 0,C 180,E1 -2611.424,E2 -2611.424} C_VEL
LIN {X 0,Y 565.875,Z 631.83,A -85,B 0,C 180,E1 -2612.848,E2 -2612.848} C_VEL
LIN {X 0,Y 565.956,Z 628.441,A -85,B 0,C 180,E1 -2614.274,E2 -2614.274} C_VEL
LIN {X 0,Y 565.989,Z 623.565,A -85,B 0,C 180,E1 -2615.702,E2 -2615.702} C_VEL
LIN {X 0,Y 565.993,Z 619.041,A -85,B 0,C 180,E1 -2616.74,E2 -2616.74} C_VEL
LIN {X 0,Y 566.048,Z 612.031,A -85,B 0,C 180,E1 -2618.03,E2 -2618.03} C_VEL
LIN {X 0,Y 566.177,Z 603.552,A -85,B 0,C 180,E1 -2619.287,E2 -2619.287} C_VEL
LIN {X 0,Y 566.295,Z 594.7,A -85,B 0,C 180,E1 -2620.368,E2 -2620.368} C_VEL
LIN {X 0,Y 566.487,Z 583.981,A -85,B 0,C 180,E1 -2621.45,E2 -2621.45} C_VEL
LIN {X 0,Y 566.609,Z 573.129,A -85,B 0,C 180,E1 -2622.355,E2 -2622.355} C_VEL
LIN {X 0,Y 566.78,Z 561.241,A -85,B 0,C 180,E1 -2623.171,E2 -2623.171} C_VEL
LIN {X 0,Y 567.034,Z 548.081,A -85,B 0,C 180,E1 -2623.896,E2 -2623.896} C_VEL
LIN {X 0,Y 567.201,Z 535.012,A -85,B 0,C 180,E1 -2624.455,E2 -2624.455} C_VEL
LIN {X 0,Y 567.357,Z 521.096,A -85,B 0,C 180,E1 -2624.895,E2 -2624.895} C_VEL
LIN {X 0,Y 567.465,Z 507.079,A -85,B 0,C 180,E1 -2625.191,E2 -2625.191} C_VEL
LIN {X 0,Y 567.686,Z 377.986,A -85,B 0,C 180,E1 -2626.86,E2 -2626.86} C_VEL
LIN {X 0,Y 566.653,Z 372.273,A -85,B 0,C 180,E1 -2626.99,E2 -2626.99} C_VEL
LIN {X 0,Y 566.843,Z 354.797,A -85,B 0,C 180,E1 -2629.445,E2 -2629.445} C_VEL
LIN {X 0,Y 567.142,Z 334.392,A -85,B 0,C 180,E1 -2632.4,E2 -2632.4} C_VEL
LIN {X 0,Y 566.22,Z 328.684,A -85,B 0,C 180,E1 -2633.321,E2 -2633.321} C_VEL
LIN {X 0,Y 566.218,Z 328.576,A -85,B 0,C 180,E1 -2635.75,E2 -2635.75} C_VEL
LIN {X 0,Y 566.211,Z 328.579,A -85,B 0,C 180,E1 -2638.203,E2 -2638.203} C_VEL
LIN {X 0,Y 566.196,Z 328.578,A -85,B 0,C 180,E1 -2641.077,E2 -2641.077} C_VEL
LIN {X 0,Y 566.217,Z 328.579,A -85,B 0,C 180,E1 -2643.735,E2 -2643.735} C_VEL
LIN {X 0,Y 566.221,Z 328.577,A -85,B 0,C 180,E1 -2646.569,E2 -2646.569} C_VEL
LIN {X 0,Y 566.221,Z 328.58,A -85,B 0,C 180,E1 -2649.686,E2 -2649.686} C_VEL
LIN {X 0,Y 566.205,Z 328.576,A -85,B 0,C 180,E1 -2652.917,E2 -2652.917} C_VEL
LIN {X 0,Y 566.204,Z 328.583,A -85,B 0,C 180,E1 -2656.049,E2 -2656.049} C_VEL
LIN {X 0,Y 566.184,Z 328.579,A -85,B 0,C 180,E1 -2658.861,E2 -2658.861} C_VEL
LIN {X 0,Y 566.19,Z 328.586,A -85,B 0,C 180,E1 -2661.637,E2 -2661.637} C_VEL
LIN {X 0,Y 566.166,Z 328.583,A -85,B 0,C 180,E1 -2664.308,E2 -2664.308} C_VEL
LIN {X 0,Y 566.225,Z 328.575,A -85,B 0,C 180,E1 -2666.898,E2 -2666.898} C_VEL
LIN {X 0,Y 566.185,Z 328.586,A -85,B 0,C 180,E1 -2669.407,E2 -2669.407} C_VEL
LIN {X 0,Y 566.216,Z 328.583,A -85,B 0,C 180,E1 -2671.858,E2 -2671.858} C_VEL
LIN {X 0,Y 566.266,Z 328.736,A -85,B 0,C 180,E1 -2674.487,E2 -2674.487} C_VEL
LIN {X 0,Y 567.363,Z 335.1,A -85,B 0,C 180,E1 -2675.288,E2 -2675.288} C_VEL
LIN {X 0,Y 567.279,Z 355.386,A -85,B 0,C 180,E1 -2677.799,E2 -2677.799} C_VEL
LIN {X 0,Y 567.064,Z 372.117,A -85,B 0,C 180,E1 -2679.884,E2 -2679.884} C_VEL
LIN {X 0,Y 566.749,Z 395.655,A -85,B 0,C 180,E1 -2682.848,E2 -2682.848} C_VEL
LIN {X 0,Y 566.543,Z 419.572,A -85,B 0,C 180,E1 -2685.818,E2 -2685.818} C_VEL
LIN {X 0,Y 566.528,Z 421.359,A -85,B 0,C 180,E1 -2686.012,E2 -2686.012} C_VEL
LIN {X 0,Y 567.234,Z 428.065,A -85,B 0,C 180,E1 -2686.133,E2 -2686.133} C_VEL
LIN {X 0,Y 566.951,Z 530.402,A -85,B 0,C 180,E1 -2687.448,E2 -2687.448} C_VEL
LIN {X 0,Y 566.874,Z 543.788,A -85,B 0,C 180,E1 -2687.765,E2 -2687.765} C_VEL
LIN {X 0,Y 566.749,Z 555.904,A -85,B 0,C 180,E1 -2688.194,E2 -2688.194} C_VEL
LIN {X 0,Y 566.644,Z 568.038,A -85,B 0,C 180,E1 -2688.776,E2 -2688.776} C_VEL
LIN {X 0,Y 566.445,Z 579.085,A -85,B 0,C 180,E1 -2689.455,E2 -2689.455} C_VEL
LIN {X 0,Y 566.315,Z 589.581,A -85,B 0,C 180,E1 -2690.265,E2 -2690.265} C_VEL
LIN {X 0,Y 566.184,Z 599.894,A -85,B 0,C 180,E1 -2691.254,E2 -2691.254} C_VEL
LIN {X 0,Y 566.081,Z 608.857,A -85,B 0,C 180,E1 -2692.33,E2 -2692.33} C_VEL
LIN {X 0,Y 566.01,Z 615.949,A -85,B 0,C 180,E1 -2693.386,E2 -2693.386} C_VEL
LIN {X 0,Y 566.004,Z 620.957,A -85,B 0,C 180,E1 -2694.299,E2 -2694.299} C_VEL
LIN {X 0,Y 565.933,Z 625.695,A -85,B 0,C 180,E1 -2695.37,E2 -2695.37} C_VEL
LIN {X 0,Y 565.928,Z 629.325,A -85,B 0,C 180,E1 -2696.44,E2 -2696.44} C_VEL
LIN {X 0,Y 565.878,Z 631.195,A -85,B 0,C 180,E1 -2697.153,E2 -2697.153} C_VEL
LIN {X 0,Y 565.839,Z 632.629,A -85,B 0,C 180,E1 -2697.865,E2 -2697.865} C_VEL
LIN {X 0,Y 565.841,Z 634.255,A -85,B 0,C 180,E1 -2699.288,E2 -2699.288} C_VEL
LIN {X 0,Y 565.839,Z 634.496,A -85,B 0,C 180,E1 -2700,E2 -2700} C_VEL
LIN {X 0,Y 565.841,Z 634.314,A -85,B 0,C 180,E1 -2700.712,E2 -2700.712} C_VEL
LIN {X 0,Y 565.838,Z 632.769,A -85,B 0,C 180,E1 -2702.135,E2 -2702.135} C_VEL
LIN {X 0,Y 565.879,Z 631.409,A -85,B 0,C 180,E1 -2702.848,E2 -2702.848} C_VEL
LIN {X 0,Y 565.927,Z 628.537,A -85,B 0,C 180,E1 -2703.917,E2 -2703.917} C_VEL
LIN {X 0,Y 565.878,Z 624.638,A -85,B 0,C 180,E1 -2704.988,E2 -2704.988} C_VEL
LIN {X 0,Y 565.988,Z 619.605,A -85,B 0,C 180,E1 -2706.059,E2 -2706.059} C_VEL
LIN {X 0,Y 566.033,Z 613.258,A -85,B 0,C 180,E1 -2707.132,E2 -2707.132} C_VEL
LIN {X 0,Y 566.128,Z 605.36,A -85,B 0,C 180,E1 -2708.208,E2 -2708.208} C_VEL
LIN {X 0,Y 566.229,Z 597.292,A -85,B 0,C 180,E1 -2709.106,E2 -2709.106} C_VEL
LIN {X 0,Y 566.333,Z 587.441,A -85,B 0,C 180,E1 -2710.005,E2 -2710.005} C_VEL
LIN {X 0,Y 566.514,Z 576.481,A -85,B 0,C 180,E1 -2710.808,E2 -2710.808} C_VEL
LIN {X 0,Y 566.662,Z 565.573,A -85,B 0,C 180,E1 -2711.446,E2 -2711.446} C_VEL
LIN {X 0,Y 566.77,Z 554.09,A -85,B 0,C 180,E1 -2711.97,E2 -2711.97} C_VEL
LIN {X 0,Y 566.91,Z 540.531,A -85,B 0,C 180,E1 -2712.416,E2 -2712.416} C_VEL
LIN {X 0,Y 567.019,Z 527.681,A -85,B 0,C 180,E1 -2712.687,E2 -2712.687} C_VEL
LIN {X 0,Y 567.19,Z 430.818,A -85,B 0,C 180,E1 -2713.923,E2 -2713.923} C_VEL
LIN {X 0,Y 566.626,Z 427.617,A -85,B 0,C 180,E1 -2713.998,E2 -2713.998} C_VEL
LIN {X 0,Y 564.682,Z 423.69,A -85,B 0,C 180,E1 -2714.186,E2 -2714.186} C_VEL
LIN {X 0,Y 561.322,Z 418.954,A -85,B 0,C 180,E1 -2714.576,E2 -2714.576} C_VEL
LIN {X 0,Y 559.75,Z 415.856,A -85,B 0,C 180,E1 -2714.922,E2 -2714.922} C_VEL
LIN {X 0,Y 559.572,Z 414.536,A -85,B 0,C 180,E1 -2715.084,E2 -2715.084} C_VEL
LIN {X 0,Y 559.909,Z 390.621,A -85,B 0,C 180,E1 -2718.099,E2 -2718.099} C_VEL
LIN {X 0,Y 560.239,Z 366.625,A -85,B 0,C 180,E1 -2721.141,E2 -2721.141} C_VEL
LIN {X 0,Y 560.567,Z 343.946,A -85,B 0,C 180,E1 -2724.006,E2 -2724.006} C_VEL
LIN {X 0,Y 560.472,Z 335.882,A -85,B 0,C 180,E1 -2725.037,E2 -2725.037} C_VEL
LIN {X 0,Y 559.2,Z 329.561,A -85,B 0,C 180,E1 -2725.933,E2 -2725.933} C_VEL
LIN {X 0,Y 559.168,Z 329.462,A -85,B 0,C 180,E1 -2728.53,E2 -2728.53} C_VEL
LIN {X 0,Y 559.151,Z 329.456,A -85,B 0,C 180,E1 -2731.273,E2 -2731.273} C_VEL
LIN {X 0,Y 559.171,Z 329.456,A -85,B 0,C 180,E1 -2733.949,E2 -2733.949} C_VEL
LIN {X 0,Y 559.145,Z 329.456,A -85,B 0,C 180,E1 -2737.108,E2 -2737.108} C_VEL
LIN {X 0,Y 559.165,Z 329.457,A -85,B 0,C 180,E1 -2739.941,E2 -2739.941} C_VEL
LIN {X 0,Y 559.163,Z 329.454,A -85,B 0,C 180,E1 -2742.743,E2 -2742.743} C_VEL
LIN {X 0,Y 559.154,Z 329.453,A -85,B 0,C 180,E1 -2745.761,E2 -2745.761} C_VEL
LIN {X 0,Y 559.167,Z 329.46,A -85,B 0,C 180,E1 -2748.229,E2 -2748.229} C_VEL
LIN {X 0,Y 559.18,Z 329.45,A -85,B 0,C 180,E1 -2751.191,E2 -2751.191} C_VEL
LIN {X 0,Y 559.163,Z 329.459,A -85,B 0,C 180,E1 -2753.79,E2 -2753.79} C_VEL
LIN {X 0,Y 559.169,Z 329.455,A -85,B 0,C 180,E1 -2756.425,E2 -2756.425} C_VEL
LIN {X 0,Y 559.161,Z 329.454,A -85,B 0,C 180,E1 -2758.98,E2 -2758.98} C_VEL
LIN {X 0,Y 559.174,Z 329.451,A -85,B 0,C 180,E1 -2761.618,E2 -2761.618} C_VEL
LIN {X 0,Y 559.186,Z 329.453,A -85,B 0,C 180,E1 -2763.902,E2 -2763.902} C_VEL
LIN {X 0,Y 559.186,Z 329.669,A -85,B 0,C 180,E1 -2766.587,E2 -2766.587} C_VEL
LIN {X 0,Y 560.224,Z 335.397,A -85,B 0,C 180,E1 -2767.503,E2 -2767.503} C_VEL
LIN {X 0,Y 559.904,Z 355.194,A -85,B 0,C 180,E1 -2770.407,E2 -2770.407} C_VEL
LIN {X 0,Y 559.673,Z 372.068,A -85,B 0,C 180,E1 -2772.819,E2 -2772.819} C_VEL
LIN {X 0,Y 560.255,Z 375.578,A -85,B 0,C 180,E1 -2772.923,E2 -2772.923} C_VEL
LIN {X 0,Y 561.01,Z 380.768,A -85,B 0,C 180,E1 -2773.015,E2 -2773.015} C_VEL
LIN {X 0,Y 560.594,Z 508.243,A -85,B 0,C 180,E1 -2774.688,E2 -2774.688} C_VEL
LIN {X 0,Y 560.482,Z 520.018,A -85,B 0,C 180,E1 -2774.941,E2 -2774.941} C_VEL
LIN {X 0,Y 560.363,Z 531.058,A -85,B 0,C 180,E1 -2775.273,E2 -2775.273} C_VEL
LIN {X 0,Y 560.205,Z 542.007,A -85,B 0,C 180,E1 -2775.7,E2 -2775.7} C_VEL
LIN {X 0,Y 560.034,Z 552.416,A -85,B 0,C 180,E1 -2776.205,E2 -2776.205} C_VEL
LIN {X 0,Y 559.824,Z 563.348,A -85,B 0,C 180,E1 -2776.847,E2 -2776.847} C_VEL
LIN {X 0,Y 559.6,Z 576.087,A -85,B 0,C 180,E1 -2777.764,E2 -2777.764} C_VEL
LIN {X 0,Y 559.405,Z 587.204,A -85,B 0,C 180,E1 -2778.76,E2 -2778.76} C_VEL
LIN {X 0,Y 559.24,Z 595.866,A -85,B 0,C 180,E1 -2779.683,E2 -2779.683} C_VEL
LIN {X 0,Y 559.122,Z 603.179,A -85,B 0,C 180,E1 -2780.595,E2 -2780.595} C_VEL
LIN {X 0,Y 559.008,Z 610.593,A -85,B 0,C 180,E1 -2781.686,E2 -2781.686} C_VEL
LIN {X 0,Y 558.908,Z 616.781,A -85,B 0,C 180,E1 -2782.775,E2 -2782.775} C_VEL
LIN {X 0,Y 558.887,Z 621.88,A -85,B 0,C 180,E1 -2783.863,E2 -2783.863} C_VEL
LIN {X 0,Y 558.821,Z 627.251,A -85,B 0,C 180,E1 -2785.31,E2 -2785.31} C_VEL
LIN {X 0,Y 558.826,Z 630.211,A -85,B 0,C 180,E1 -2786.394,E2 -2786.394} C_VEL
LIN {X 0,Y 558.745,Z 632.945,A -85,B 0,C 180,E1 -2787.837,E2 -2787.837} C_VEL
LIN {X 0,Y 558.737,Z 634.266,A -85,B 0,C 180,E1 -2789.278,E2 -2789.278} C_VEL
LIN {X 0,Y 558.739,Z 634.496,A -85,B 0,C 180,E1 -2789.999,E2 -2789.999} C_VEL
LIN {X 0,Y 558.741,Z 633.855,A -85,B 0,C 180,E1 -2791.441,E2 -2791.441} C_VEL
LIN {X 0,Y 558.794,Z 631.876,A -85,B 0,C 180,E1 -2792.883,E2 -2792.883} C_VEL
LIN {X 0,Y 558.826,Z 630.436,A -85,B 0,C 180,E1 -2793.604,E2 -2793.604} C_VEL
LIN {X 0,Y 558.791,Z 626.33,A -85,B 0,C 180,E1 -2795.05,E2 -2795.05} C_VEL
LIN {X 0,Y 558.883,Z 622.277,A -85,B 0,C 180,E1 -2796.135,E2 -2796.135} C_VEL
LIN {X 0,Y 558.905,Z 617.262,A -85,B 0,C 180,E1 -2797.223,E2 -2797.223} C_VEL
LIN {X 0,Y 559.006,Z 611.163,A -85,B 0,C 180,E1 -2798.312,E2 -2798.312} C_VEL
LIN {X 0,Y 559.105,Z 603.849,A -85,B 0,C 180,E1 -2799.404,E2 -2799.404} C_VEL
LIN {X 0,Y 559.264,Z 595.092,A -85,B 0,C 180,E1 -2800.498,E2 -2800.498} C_VEL
LIN {X 0,Y 559.453,Z 584.51,A -85,B 0,C 180,E1 -2801.594,E2 -2801.594} C_VEL
LIN {X 0,Y 559.63,Z 573.713,A -85,B 0,C 180,E1 -2802.51,E2 -2802.51} C_VEL
LIN {X 0,Y 559.8,Z 563.34,A -85,B 0,C 180,E1 -2803.244,E2 -2803.244} C_VEL
LIN {X 0,Y 560.02,Z 552.403,A -85,B 0,C 180,E1 -2803.886,E2 -2803.886} C_VEL
LIN {X 0,Y 560.174,Z 541.986,A -85,B 0,C 180,E1 -2804.392,E2 -2804.392} C_VEL
LIN {X 0,Y 560.381,Z 530.336,A -85,B 0,C 180,E1 -2804.841,E2 -2804.841} C_VEL
LIN {X 0,Y 560.505,Z 519.082,A -85,B 0,C 180,E1 -2805.172,E2 -2805.172} C_VEL
LIN {X 0,Y 560.601,Z 506.812,A -85,B 0,C 180,E1 -2805.426,E2 -2805.426} C_VEL
LIN {X 0,Y 560.948,Z 379.163,A -85,B 0,C 180,E1 -2807.098,E2 -2807.098} C_VEL
LIN {X 0,Y 559.73,Z 372.473,A -85,B 0,C 180,E1 -2807.242,E2 -2807.242} C_VEL
LIN {X 0,Y 559.66,Z 370.023,A -85,B 0,C 180,E1 -2807.54,E2 -2807.54} C_VEL
LIN {X 0,Y 559.966,Z 350.403,A -85,B 0,C 180,E1 -2810.381,E2 -2810.381} C_VEL
LIN {X 0,Y 560.2,Z 334.707,A -85,B 0,C 180,E1 -2812.691,E2 -2812.691} C_VEL
LIN {X 0,Y 559.183,Z 329.575,A -85,B 0,C 180,E1 -2813.534,E2 -2813.534} C_VEL
LIN {X 0,Y 559.197,Z 329.451,A -85,B 0,C 180,E1 -2816.095,E2 -2816.095} C_VEL
LIN {X 0,Y 559.164,Z 329.451,A -85,B 0,C 180,E1 -2818.528,E2 -2818.528} C_VEL
LIN {X 0,Y 559.154,Z 329.455,A -85,B 0,C 180,E1 -2821.274,E2 -2821.274} C_VEL
LIN {X 0,Y 559.176,Z 329.458,A -85,B 0,C 180,E1 -2823.95,E2 -2823.95} C_VEL
LIN {X 0,Y 559.166,Z 329.456,A -85,B 0,C 180,E1 -2826.448,E2 -2826.448} C_VEL
LIN {X 0,Y 559.175,Z 329.451,A -85,B 0,C 180,E1 -2828.932,E2 -2828.932} C_VEL
LIN {X 0,Y 559.187,Z 329.456,A -85,B 0,C 180,E1 -2831.766,E2 -2831.766} C_VEL
LIN {X 0,Y 559.134,Z 329.453,A -85,B 0,C 180,E1 -2834.738,E2 -2834.738} C_VEL
LIN {X 0,Y 559.167,Z 329.453,A -85,B 0,C 180,E1 -2837.257,E2 -2837.257} C_VEL
LIN {X 0,Y 559.18,Z 329.452,A -85,B 0,C 180,E1 -2840.134,E2 -2840.134} C_VEL
LIN {X 0,Y 559.139,Z 329.45,A -85,B 0,C 180,E1 -2842.891,E2 -2842.891} C_VEL
LIN {X 0,Y 559.153,Z 329.461,A -85,B 0,C 180,E1 -2845.555,E2 -2845.555} C_VEL
LIN {X 0,Y 559.165,Z 329.453,A -85,B 0,C 180,E1 -2848.137,E2 -2848.137} C_VEL
LIN {X 0,Y 559.15,Z 329.446,A -85,B 0,C 180,E1 -2850.647,E2 -2850.647} C_VEL
LIN {X 0,Y 559.174,Z 329.451,A -85,B 0,C 180,E1 -2853.169,E2 -2853.169} C_VEL
LIN {X 0,Y 559.152,Z 329.464,A -85,B 0,C 180,E1 -2855.495,E2 -2855.495} C_VEL
LIN {X 0,Y 559.155,Z 329.451,A -85,B 0,C 180,E1 -2858.447,E2 -2858.447} C_VEL
LIN {X 0,Y 559.163,Z 329.455,A -85,B 0,C 180,E1 -2860.926,E2 -2860.926} C_VEL
LIN {X 0,Y 559.165,Z 329.451,A -85,B 0,C 180,E1 -2863.948,E2 -2863.948} C_VEL
LIN {X 0,Y 559.166,Z 329.452,A -85,B 0,C 180,E1 -2866.184,E2 -2866.184} C_VEL
LIN {X 0,Y 559.226,Z 329.453,A -85,B 0,C 180,E1 -2869.134,E2 -2869.134} C_VEL
LIN {X 0,Y 559.205,Z 329.447,A -85,B 0,C 180,E1 -2872.054,E2 -2872.054} C_VEL
LIN {X 0,Y 559.252,Z 329.448,A -85,B 0,C 180,E1 -2874.953,E2 -2874.953} C_VEL
LIN {X 0,Y 559.244,Z 329.442,A -85,B 0,C 180,E1 -2877.839,E2 -2877.839} C_VEL
LIN {X 0,Y 559.271,Z 329.445,A -85,B 0,C 180,E1 -2880.72,E2 -2880.72} C_VEL
LIN {X 0,Y 559.239,Z 329.45,A -85,B 0,C 180,E1 -2882.881,E2 -2882.881} C_VEL
LIN {X 0,Y 559.223,Z 329.445,A -85,B 0,C 180,E1 -2885.77,E2 -2885.77} C_VEL
LIN {X 0,Y 559.196,Z 329.455,A -85,B 0,C 180,E1 -2888.674,E2 -2888.674} C_VEL
LIN {X 0,Y 559.199,Z 329.448,A -85,B 0,C 180,E1 -2891.601,E2 -2891.601} C_VEL
LIN {X 0,Y 559.188,Z 329.456,A -85,B 0,C 180,E1 -2894.596,E2 -2894.596} C_VEL
LIN {X 0,Y 559.156,Z 329.453,A -85,B 0,C 180,E1 -2897.557,E2 -2897.557} C_VEL
LIN {X 0,Y 559.166,Z 329.452,A -85,B 0,C 180,E1 -2899.838,E2 -2899.838} C_VEL
LIN {X 0,Y 559.147,Z 329.455,A -85,B 0,C 180,E1 -2902.153,E2 -2902.153} C_VEL
LIN {X 0,Y 559.152,Z 329.463,A -85,B 0,C 180,E1 -2904.505,E2 -2904.505} C_VEL
LIN {X 0,Y 559.17,Z 329.451,A -85,B 0,C 180,E1 -2906.902,E2 -2906.902} C_VEL
LIN {X 0,Y 559.141,Z 329.449,A -85,B 0,C 180,E1 -2909.859,E2 -2909.859} C_VEL
LIN {X 0,Y 559.168,Z 329.457,A -85,B 0,C 180,E1 -2912.714,E2 -2912.714} C_VEL
LIN {X 0,Y 559.149,Z 329.454,A -85,B 0,C 180,E1 -2915.323,E2 -2915.323} C_VEL
LIN {X 0,Y 559.127,Z 329.457,A -85,B 0,C 180,E1 -2918.018,E2 -2918.018} C_VEL
LIN {X 0,Y 559.173,Z 329.454,A -85,B 0,C 180,E1 -2920.811,E2 -2920.811} C_VEL
LIN {X 0,Y 559.158,Z 329.455,A -85,B 0,C 180,E1 -2923.732,E2 -2923.732} C_VEL
LIN {X 0,Y 559.161,Z 329.454,A -85,B 0,C 180,E1 -2926.802,E2 -2926.802} C_VEL
LIN {X 0,Y 559.171,Z 329.451,A -85,B 0,C 180,E1 -2929.191,E2 -2929.191} C_VEL
LIN {X 0,Y 559.131,Z 329.465,A -85,B 0,C 180,E1 -2931.984,E2 -2931.984} C_VEL
LIN {X 0,Y 559.157,Z 329.454,A -85,B 0,C 180,E1 -2934.784,E2 -2934.784} C_VEL
LIN {X 0,Y 559.171,Z 329.453,A -85,B 0,C 180,E1 -2937.362,E2 -2937.362} C_VEL
LIN {X 0,Y 559.187,Z 329.449,A -85,B 0,C 180,E1 -2940.136,E2 -2940.136} C_VEL
LIN {X 0,Y 559.18,Z 329.454,A -85,B 0,C 180,E1 -2943.171,E2 -2943.171} C_VEL
LIN {X 0,Y 559.156,Z 329.462,A -85,B 0,C 180,E1 -2945.496,E2 -2945.496} C_VEL
LIN {X 0,Y 559.181,Z 329.645,A -85,B 0,C 180,E1 -2946.533,E2 -2946.533} C_VEL
LIN {X 0,Y 560.267,Z 335.712,A -85,B 0,C 180,E1 -2947.507,E2 -2947.507} C_VEL
LIN {X 0,Y 559.878,Z 357.023,A -85,B 0,C 180,E1 -2950.628,E2 -2950.628} C_VEL
LIN {X 0,Y 559.7,Z 372.047,A -85,B 0,C 180,E1 -2952.773,E2 -2952.773} C_VEL
LIN {X 0,Y 560.179,Z 375.236,A -85,B 0,C 180,E1 -2952.871,E2 -2952.871} C_VEL
LIN {X 0,Y 560.992,Z 379.889,A -85,B 0,C 180,E1 -2952.958,E2 -2952.958} C_VEL
LIN {X 0,Y 560.618,Z 508.698,A -85,B 0,C 180,E1 -2954.644,E2 -2954.644} C_VEL
LIN {X 0,Y 560.441,Z 523,A -85,B 0,C 180,E1 -2954.969,E2 -2954.969} C_VEL
LIN {X 0,Y 560.301,Z 536.499,A -85,B 0,C 180,E1 -2955.422,E2 -2955.422} C_VEL
LIN {X 0,Y 560.105,Z 549.895,A -85,B 0,C 180,E1 -2956.023,E2 -2956.023} C_VEL
LIN {X 0,Y 559.838,Z 562.695,A -85,B 0,C 180,E1 -2956.757,E2 -2956.757} C_VEL
LIN {X 0,Y 559.647,Z 574.324,A -85,B 0,C 180,E1 -2957.582,E2 -2957.582} C_VEL
LIN {X 0,Y 559.429,Z 584.928,A -85,B 0,C 180,E1 -2958.493,E2 -2958.493} C_VEL
LIN {X 0,Y 559.272,Z 594.716,A -85,B 0,C 180,E1 -2959.502,E2 -2959.502} C_VEL
LIN {X 0,Y 559.12,Z 603.565,A -85,B 0,C 180,E1 -2960.596,E2 -2960.596} C_VEL
LIN {X 0,Y 558.985,Z 612.042,A -85,B 0,C 180,E1 -2961.87,E2 -2961.87} C_VEL
LIN {X 0,Y 558.901,Z 618.87,A -85,B 0,C 180,E1 -2963.14,E2 -2963.14} C_VEL
LIN {X 0,Y 558.912,Z 623.572,A -85,B 0,C 180,E1 -2964.228,E2 -2964.228} C_VEL
LIN {X 0,Y 558.865,Z 628.449,A -85,B 0,C 180,E1 -2965.674,E2 -2965.674} C_VEL
LIN {X 0,Y 558.796,Z 631.836,A -85,B 0,C 180,E1 -2967.117,E2 -2967.117} C_VEL
LIN {X 0,Y 558.74,Z 633.835,A -85,B 0,C 180,E1 -2968.559,E2 -2968.559} C_VEL
LIN {X 0,Y 558.738,Z 634.5,A -85,B 0,C 180,E1 -2970.001,E2 -2970.001} C_VEL
LIN {X 0,Y 558.74,Z 633.833,A -85,B 0,C 180,E1 -2971.442,E2 -2971.442} C_VEL
LIN {X 0,Y 558.796,Z 631.83,A -85,B 0,C 180,E1 -2972.885,E2 -2972.885} C_VEL
LIN {X 0,Y 558.865,Z 628.441,A -85,B 0,C 180,E1 -2974.328,E2 -2974.328} C_VEL
LIN {X 0,Y 558.917,Z 623.565,A -85,B 0,C 180,E1 -2975.774,E2 -2975.774} C_VEL
LIN {X 0,Y 558.903,Z 618.861,A -85,B 0,C 180,E1 -2976.861,E2 -2976.861} C_VEL
LIN {X 0,Y 558.987,Z 612.03,A -85,B 0,C 180,E1 -2978.132,E2 -2978.132} C_VEL
LIN {X 0,Y 559.118,Z 603.551,A -85,B 0,C 180,E1 -2979.406,E2 -2979.406} C_VEL
LIN {X 0,Y 559.273,Z 594.699,A -85,B 0,C 180,E1 -2980.499,E2 -2980.499} C_VEL
LIN {X 0,Y 559.489,Z 583.979,A -85,B 0,C 180,E1 -2981.595,E2 -2981.595} C_VEL
LIN {X 0,Y 559.64,Z 573.127,A -85,B 0,C 180,E1 -2982.512,E2 -2982.512} C_VEL
LIN {X 0,Y 559.843,Z 561.238,A -85,B 0,C 180,E1 -2983.337,E2 -2983.337} C_VEL
LIN {X 0,Y 560.133,Z 548.082,A -85,B 0,C 180,E1 -2984.07,E2 -2984.07} C_VEL
LIN {X 0,Y 560.328,Z 535.232,A -85,B 0,C 180,E1 -2984.628,E2 -2984.628} C_VEL
LIN {X 0,Y 560.471,Z 520.97,A -85,B 0,C 180,E1 -2985.085,E2 -2985.085} C_VEL
LIN {X 0,Y 560.63,Z 507.078,A -85,B 0,C 180,E1 -2985.38,E2 -2985.38} C_VEL
LIN {X 0,Y 560.916,Z 379.003,A -85,B 0,C 180,E1 -2987.056,E2 -2987.056} C_VEL
LIN {X 0,Y 559.675,Z 372.293,A -85,B 0,C 180,E1 -2987.209,E2 -2987.209} C_VEL
LIN {X 0,Y 559.759,Z 364.467,A -85,B 0,C 180,E1 -2988.294,E2 -2988.294} C_VEL
LIN {X 0,Y 560.077,Z 344.853,A -85,B 0,C 180,E1 -2991.148,E2 -2991.148} C_VEL
LIN {X 0,Y 560.16,Z 334.392,A -85,B 0,C 180,E1 -2992.694,E2 -2992.694} C_VEL
LIN {X 0,Y 559.183,Z 329.572,A -85,B 0,C 180,E1 -2993.49,E2 -2993.49} C_VEL
LIN {X 0,Y 559.185,Z 329.454,A -85,B 0,C 180,E1 -2996.098,E2 -2996.098} C_VEL
LIN {X 0,Y 559.169,Z 329.453,A -85,B 0,C 180,E1 -2998.53,E2 -2998.53} C_VEL
LIN {X 0,Y 559.151,Z 329.456,A -85,B 0,C 180,E1 -3001.274,E2 -3001.274} C_VEL
LIN {X 0,Y 559.173,Z 329.46,A -85,B 0,C 180,E1 -3003.95,E2 -3003.95} C_VEL
LIN {X 0,Y 559.174,Z 329.456,A -85,B 0,C 180,E1 -3006.449,E2 -3006.449} C_VEL
LIN {X 0,Y 559.179,Z 329.452,A -85,B 0,C 180,E1 -3008.934,E2 -3008.934} C_VEL
LIN {X 0,Y 559.167,Z 329.46,A -85,B 0,C 180,E1 -3011.771,E2 -3011.771} C_VEL
LIN {X 0,Y 559.143,Z 329.456,A -85,B 0,C 180,E1 -3014.74,E2 -3014.74} C_VEL
LIN {X 0,Y 559.179,Z 329.46,A -85,B 0,C 180,E1 -3017.863,E2 -3017.863} C_VEL
LIN {X 0,Y 559.178,Z 329.453,A -85,B 0,C 180,E1 -3021.066,E2 -3021.066} C_VEL
LIN {X 0,Y 559.143,Z 329.465,A -85,B 0,C 180,E1 -3023.789,E2 -3023.789} C_VEL
LIN {X 0,Y 559.167,Z 329.455,A -85,B 0,C 180,E1 -3026.425,E2 -3026.425} C_VEL
LIN {X 0,Y 559.159,Z 329.456,A -85,B 0,C 180,E1 -3028.981,E2 -3028.981} C_VEL
LIN {X 0,Y 559.173,Z 329.461,A -85,B 0,C 180,E1 -3031.619,E2 -3031.619} C_VEL
LIN {X 0,Y 559.228,Z 329.668,A -85,B 0,C 180,E1 -3034.388,E2 -3034.388} C_VEL
LIN {X 0,Y 560.423,Z 337.423,A -85,B 0,C 180,E1 -3035.356,E2 -3035.356} C_VEL
LIN {X 0,Y 560.247,Z 357.725,A -85,B 0,C 180,E1 -3037.893,E2 -3037.893} C_VEL
LIN {X 0,Y 560.072,Z 376.826,A -85,B 0,C 180,E1 -3040.243,E2 -3040.243} C_VEL
LIN {X 0,Y 559.767,Z 399.138,A -85,B 0,C 180,E1 -3043.069,E2 -3043.069} C_VEL
LIN {X 0,Y 559.542,Z 421.372,A -85,B 0,C 180,E1 -3045.834,E2 -3045.834} C_VEL
LIN {X 0,Y 560.332,Z 428.11,A -85,B 0,C 180,E1 -3045.959,E2 -3045.959} C_VEL
LIN {X 0,Y 560.041,Z 530.421,A -85,B 0,C 180,E1 -3047.291,E2 -3047.291} C_VEL
LIN {X 0,Y 559.922,Z 543.816,A -85,B 0,C 180,E1 -3047.611,E2 -3047.611} C_VEL
LIN {X 0,Y 559.799,Z 555.91,A -85,B 0,C 180,E1 -3048.045,E2 -3048.045} C_VEL
LIN {X 0,Y 559.654,Z 568.614,A -85,B 0,C 180,E1 -3048.665,E2 -3048.665} C_VEL
LIN {X 0,Y 559.432,Z 580.371,A -85,B 0,C 180,E1 -3049.413,E2 -3049.413} C_VEL
LIN {X 0,Y 559.262,Z 591.648,A -85,B 0,C 180,E1 -3050.324,E2 -3050.324} C_VEL
LIN {X 0,Y 559.144,Z 601.525,A -85,B 0,C 180,E1 -3051.325,E2 -3051.325} C_VEL
LIN {X 0,Y 558.998,Z 610.176,A -85,B 0,C 180,E1 -3052.414,E2 -3052.414} C_VEL
LIN {X 0,Y 558.895,Z 617.128,A -85,B 0,C 180,E1 -3053.502,E2 -3053.502} C_VEL
LIN {X 0,Y 558.869,Z 622.677,A -85,B 0,C 180,E1 -3054.588,E2 -3054.588} C_VEL
LIN {X 0,Y 558.869,Z 627.031,A -85,B 0,C 180,E1 -3055.673,E2 -3055.673} C_VEL
LIN {X 0,Y 558.837,Z 629.326,A -85,B 0,C 180,E1 -3056.395,E2 -3056.395} C_VEL
LIN {X 0,Y 558.8,Z 631.195,A -85,B 0,C 180,E1 -3057.116,E2 -3057.116} C_VEL
LIN {X 0,Y 558.745,Z 632.63,A -85,B 0,C 180,E1 -3057.838,E2 -3057.838} C_VEL
LIN {X 0,Y 558.742,Z 634.255,A -85,B 0,C 180,E1 -3059.279,E2 -3059.279} C_VEL
LIN {X 0,Y 558.74,Z 634.496,A -85,B 0,C 180,E1 -3060,E2 -3060} C_VEL
LIN {X 0,Y 558.741,Z 634.313,A -85,B 0,C 180,E1 -3060.721,E2 -3060.721} C_VEL
LIN {X 0,Y 558.745,Z 632.768,A -85,B 0,C 180,E1 -3062.163,E2 -3062.163} C_VEL
LIN {X 0,Y 558.8,Z 631.408,A -85,B 0,C 180,E1 -3062.884,E2 -3062.884} C_VEL
LIN {X 0,Y 558.844,Z 628.536,A -85,B 0,C 180,E1 -3063.966,E2 -3063.966} C_VEL
LIN {X 0,Y 558.798,Z 624.637,A -85,B 0,C 180,E1 -3065.051,E2 -3065.051} C_VEL
LIN {X 0,Y 558.908,Z 619.602,A -85,B 0,C 180,E1 -3066.136,E2 -3066.136} C_VEL
LIN {X 0,Y 558.975,Z 612.052,A -85,B 0,C 180,E1 -3067.405,E2 -3067.405} C_VEL
LIN {X 0,Y 559.105,Z 603.875,A -85,B 0,C 180,E1 -3068.494,E2 -3068.494} C_VEL
LIN {X 0,Y 559.223,Z 595.473,A -85,B 0,C 180,E1 -3069.403,E2 -3069.403} C_VEL
LIN {X 0,Y 559.398,Z 585.172,A -85,B 0,C 180,E1 -3070.313,E2 -3070.313} C_VEL
LIN {X 0,Y 559.584,Z 574.161,A -85,B 0,C 180,E1 -3071.095,E2 -3071.095} C_VEL
LIN {X 0,Y 559.712,Z 562.628,A -85,B 0,C 180,E1 -3071.739,E2 -3071.739} C_VEL
LIN {X 0,Y 559.887,Z 550.116,A -85,B 0,C 180,E1 -3072.271,E2 -3072.271} C_VEL
LIN {X 0,Y 559.987,Z 536.895,A -85,B 0,C 180,E1 -3072.664,E2 -3072.664} C_VEL
LIN {X 0,Y 560.095,Z 522.717,A -85,B 0,C 180,E1 -3072.915,E2 -3072.915} C_VEL
LIN {X 0,Y 560.161,Z 426.109,A -85,B 0,C 180,E1 -3074.162,E2 -3074.162} C_VEL
LIN {X 0,Y 559.52,Z 421.152,A -85,B 0,C 180,E1 -3074.271,E2 -3074.271} C_VEL
LIN {X 0,Y 559.572,Z 414.536,A -85,B 0,C 180,E1 -3075.084,E2 -3075.084} C_VEL
LIN {X 0,Y 558.972,Z 410.911,A -85,B 0,C 180,E1 -3075.558,E2 -3075.558} C_VEL
LIN {X 0,Y 553.43,Z 399.701,A -85,B 0,C 180,E1 -3077.147,E2 -3077.147} C_VEL
LIN {X 0,Y 552.844,Z 396.03,A -85,B 0,C 180,E1 -3077.627,E2 -3077.627} C_VEL
LIN {X 0,Y 553.2,Z 373.886,A -85,B 0,C 180,E1 -3080.449,E2 -3080.449} C_VEL
LIN {X 0,Y 553.557,Z 350.961,A -85,B 0,C 180,E1 -3083.37,E2 -3083.37} C_VEL
LIN {X 0,Y 553.673,Z 338.579,A -85,B 0,C 180,E1 -3084.959,E2 -3084.959} C_VEL
LIN {X 0,Y 552.172,Z 330.463,A -85,B 0,C 180,E1 -3086.098,E2 -3086.098} C_VEL
LIN {X 0,Y 552.115,Z 330.337,A -85,B 0,C 180,E1 -3088.928,E2 -3088.928} C_VEL
LIN {X 0,Y 552.116,Z 330.332,A -85,B 0,C 180,E1 -3091.475,E2 -3091.475} C_VEL
LIN {X 0,Y 552.138,Z 330.335,A -85,B 0,C 180,E1 -3094.17,E2 -3094.17} C_VEL
LIN {X 0,Y 552.11,Z 330.336,A -85,B 0,C 180,E1 -3096.747,E2 -3096.747} C_VEL
LIN {X 0,Y 552.134,Z 330.329,A -85,B 0,C 180,E1 -3099.527,E2 -3099.527} C_VEL
LIN {X 0,Y 552.135,Z 330.334,A -85,B 0,C 180,E1 -3102.425,E2 -3102.425} C_VEL
LIN {X 0,Y 552.098,Z 330.33,A -85,B 0,C 180,E1 -3105.562,E2 -3105.562} C_VEL
LIN {X 0,Y 552.125,Z 330.332,A -85,B 0,C 180,E1 -3108.554,E2 -3108.554} C_VEL
LIN {X 0,Y 552.123,Z 330.33,A -85,B 0,C 180,E1 -3111.411,E2 -3111.411} C_VEL
LIN {X 0,Y 552.107,Z 330.338,A -85,B 0,C 180,E1 -3114.157,E2 -3114.157} C_VEL
LIN {X 0,Y 552.121,Z 330.33,A -85,B 0,C 180,E1 -3116.814,E2 -3116.814} C_VEL
LIN {X 0,Y 552.108,Z 330.335,A -85,B 0,C 180,E1 -3119.39,E2 -3119.39} C_VEL
LIN {X 0,Y 552.126,Z 330.333,A -85,B 0,C 180,E1 -3121.902,E2 -3121.902} C_VEL
LIN {X 0,Y 552.161,Z 330.326,A -85,B 0,C 180,E1 -3124.649,E2 -3124.649} C_VEL
LIN {X 0,Y 552.117,Z 330.443,A -85,B 0,C 180,E1 -3126.369,E2 -3126.369} C_VEL
LIN {X 0,Y 553.306,Z 336.708,A -85,B 0,C 180,E1 -3127.403,E2 -3127.403} C_VEL
LIN {X 0,Y 552.987,Z 355.065,A -85,B 0,C 180,E1 -3130.132,E2 -3130.132} C_VEL
LIN {X 0,Y 552.72,Z 372.135,A -85,B 0,C 180,E1 -3132.601,E2 -3132.601} C_VEL
LIN {X 0,Y 553.413,Z 376.248,A -85,B 0,C 180,E1 -3132.714,E2 -3132.714} C_VEL
LIN {X 0,Y 554.233,Z 381.553,A -85,B 0,C 180,E1 -3132.811,E2 -3132.811} C_VEL
LIN {X 0,Y 553.751,Z 508.221,A -85,B 0,C 180,E1 -3134.495,E2 -3134.495} C_VEL
LIN {X 0,Y 553.634,Z 519.871,A -85,B 0,C 180,E1 -3134.746,E2 -3134.746} C_VEL
LIN {X 0,Y 553.501,Z 530.355,A -85,B 0,C 180,E1 -3135.062,E2 -3135.062} C_VEL
LIN {X 0,Y 553.328,Z 540.926,A -85,B 0,C 180,E1 -3135.471,E2 -3135.471} C_VEL
LIN {X 0,Y 553.188,Z 550.664,A -85,B 0,C 180,E1 -3135.937,E2 -3135.937} C_VEL
LIN {X 0,Y 552.929,Z 560.419,A -85,B 0,C 180,E1 -3136.493,E2 -3136.493} C_VEL
LIN {X 0,Y 552.744,Z 570,A -85,B 0,C 180,E1 -3137.143,E2 -3137.143} C_VEL
LIN {X 0,Y 552.541,Z 579.289,A -85,B 0,C 180,E1 -3137.884,E2 -3137.884} C_VEL
LIN {X 0,Y 552.399,Z 588.533,A -85,B 0,C 180,E1 -3138.753,E2 -3138.753} C_VEL
LIN {X 0,Y 552.236,Z 595.86,A -85,B 0,C 180,E1 -3139.551,E2 -3139.551} C_VEL
LIN {X 0,Y 552.073,Z 603.174,A -85,B 0,C 180,E1 -3140.473,E2 -3140.473} C_VEL
LIN {X 0,Y 551.963,Z 609.458,A -85,B 0,C 180,E1 -3141.395,E2 -3141.395} C_VEL
LIN {X 0,Y 551.903,Z 614.875,A -85,B 0,C 180,E1 -3142.315,E2 -3142.315} C_VEL
LIN {X 0,Y 551.824,Z 620.308,A -85,B 0,C 180,E1 -3143.417,E2 -3143.417} C_VEL
LIN {X 0,Y 551.792,Z 624.751,A -85,B 0,C 180,E1 -3144.518,E2 -3144.518} C_VEL
LIN {X 0,Y 551.76,Z 628.305,A -85,B 0,C 180,E1 -3145.616,E2 -3145.616} C_VEL
LIN {X 0,Y 551.741,Z 630.214,A -85,B 0,C 180,E1 -3146.348,E2 -3146.348} C_VEL
LIN {X 0,Y 551.656,Z 632.943,A -85,B 0,C 180,E1 -3147.809,E2 -3147.809} C_VEL
LIN {X 0,Y 551.637,Z 634.259,A -85,B 0,C 180,E1 -3149.269,E2 -3149.269} C_VEL
LIN {X 0,Y 551.64,Z 634.496,A -85,B 0,C 180,E1 -3149.999,E2 -3149.999} C_VEL
LIN {X 0,Y 551.64,Z 633.851,A -85,B 0,C 180,E1 -3151.459,E2 -3151.459} C_VEL
LIN {X 0,Y 551.719,Z 631.868,A -85,B 0,C 180,E1 -3152.92,E2 -3152.92} C_VEL
LIN {X 0,Y 551.741,Z 630.436,A -85,B 0,C 180,E1 -3153.651,E2 -3153.651} C_VEL
LIN {X 0,Y 551.716,Z 626.321,A -85,B 0,C 180,E1 -3155.115,E2 -3155.115} C_VEL
LIN {X 0,Y 551.819,Z 623.772,A -85,B 0,C 180,E1 -3155.847,E2 -3155.847} C_VEL
LIN {X 0,Y 551.829,Z 617.25,A -85,B 0,C 180,E1 -3157.316,E2 -3157.316} C_VEL
LIN {X 0,Y 551.96,Z 611.152,A -85,B 0,C 180,E1 -3158.419,E2 -3158.419} C_VEL
LIN {X 0,Y 552.061,Z 605.166,A -85,B 0,C 180,E1 -3159.34,E2 -3159.34} C_VEL
LIN {X 0,Y 552.173,Z 598.186,A -85,B 0,C 180,E1 -3160.263,E2 -3160.263} C_VEL
LIN {X 0,Y 552.355,Z 589.452,A -85,B 0,C 180,E1 -3161.244,E2 -3161.244} C_VEL
LIN {X 0,Y 552.51,Z 580.33,A -85,B 0,C 180,E1 -3162.114,E2 -3162.114} C_VEL
LIN {X 0,Y 552.703,Z 571.217,A -85,B 0,C 180,E1 -3162.856,E2 -3162.856} C_VEL
LIN {X 0,Y 552.916,Z 561.853,A -85,B 0,C 180,E1 -3163.506,E2 -3163.506} C_VEL
LIN {X 0,Y 553.096,Z 552.379,A -85,B 0,C 180,E1 -3164.063,E2 -3164.063} C_VEL
LIN {X 0,Y 553.268,Z 541.95,A -85,B 0,C 180,E1 -3164.575,E2 -3164.575} C_VEL
LIN {X 0,Y 553.501,Z 531.192,A -85,B 0,C 180,E1 -3164.999,E2 -3164.999} C_VEL
LIN {X 0,Y 553.63,Z 519.943,A -85,B 0,C 180,E1 -3165.342,E2 -3165.342} C_VEL
LIN {X 0,Y 553.743,Z 509.439,A -85,B 0,C 180,E1 -3165.575,E2 -3165.575} C_VEL
LIN {X 0,Y 553.908,Z 473.905,A -85,B 0,C 180,E1 -3166.066,E2 -3166.066} C_VEL
LIN {X 0,Y 554.138,Z 380.035,A -85,B 0,C 180,E1 -3167.303,E2 -3167.303} C_VEL
LIN {X 0,Y 552.735,Z 372.412,A -85,B 0,C 180,E1 -3167.47,E2 -3167.47} C_VEL
LIN {X 0,Y 552.742,Z 368.711,A -85,B 0,C 180,E1 -3167.958,E2 -3167.958} C_VEL
LIN {X 0,Y 553.093,Z 349.091,A -85,B 0,C 180,E1 -3170.841,E2 -3170.841} C_VEL
LIN {X 0,Y 553.261,Z 336.011,A -85,B 0,C 180,E1 -3172.794,E2 -3172.794} C_VEL
LIN {X 0,Y 552.149,Z 330.401,A -85,B 0,C 180,E1 -3173.736,E2 -3173.736} C_VEL
LIN {X 0,Y 552.134,Z 330.334,A -85,B 0,C 180,E1 -3176.455,E2 -3176.455} C_VEL
LIN {X 0,Y 552.116,Z 330.324,A -85,B 0,C 180,E1 -3178.927,E2 -3178.927} C_VEL
LIN {X 0,Y 552.133,Z 330.331,A -85,B 0,C 180,E1 -3181.479,E2 -3181.479} C_VEL
LIN {X 0,Y 552.144,Z 330.336,A -85,B 0,C 180,E1 -3184.172,E2 -3184.172} C_VEL
LIN {X 0,Y 552.108,Z 330.333,A -85,B 0,C 180,E1 -3186.745,E2 -3186.745} C_VEL
LIN {X 0,Y 552.131,Z 330.331,A -85,B 0,C 180,E1 -3189.525,E2 -3189.525} C_VEL
LIN {X 0,Y 552.125,Z 330.333,A -85,B 0,C 180,E1 -3192.424,E2 -3192.424} C_VEL
LIN {X 0,Y 552.094,Z 330.334,A -85,B 0,C 180,E1 -3195.562,E2 -3195.562} C_VEL
LIN {X 0,Y 552.165,Z 330.325,A -85,B 0,C 180,E1 -3198.671,E2 -3198.671} C_VEL
LIN {X 0,Y 552.113,Z 330.332,A -85,B 0,C 180,E1 -3201.41,E2 -3201.41} C_VEL
LIN {X 0,Y 552.105,Z 330.334,A -85,B 0,C 180,E1 -3204.158,E2 -3204.158} C_VEL
LIN {X 0,Y 552.121,Z 330.331,A -85,B 0,C 180,E1 -3206.814,E2 -3206.814} C_VEL
LIN {X 0,Y 552.106,Z 330.336,A -85,B 0,C 180,E1 -3209.391,E2 -3209.391} C_VEL
LIN {X 0,Y 552.119,Z 330.329,A -85,B 0,C 180,E1 -3211.902,E2 -3211.902} C_VEL
LIN {X 0,Y 552.147,Z 330.326,A -85,B 0,C 180,E1 -3214.648,E2 -3214.648} C_VEL
LIN {X 0,Y 552.106,Z 330.338,A -85,B 0,C 180,E1 -3217.55,E2 -3217.55} C_VEL
LIN {X 0,Y 552.148,Z 330.327,A -85,B 0,C 180,E1 -3220.674,E2 -3220.674} C_VEL
LIN {X 0,Y 552.114,Z 330.331,A -85,B 0,C 180,E1 -3223.737,E2 -3223.737} C_VEL
LIN {X 0,Y 552.128,Z 330.329,A -85,B 0,C 180,E1 -3226.004,E2 -3226.004} C_VEL
LIN {X 0,Y 552.186,Z 330.327,A -85,B 0,C 180,E1 -3228.994,E2 -3228.994} C_VEL
LIN {X 0,Y 552.158,Z 330.325,A -85,B 0,C 180,E1 -3231.951,E2 -3231.951} C_VEL
LIN {X 0,Y 552.226,Z 330.323,A -85,B 0,C 180,E1 -3234.889,E2 -3234.889} C_VEL
LIN {X 0,Y 552.215,Z 330.318,A -85,B 0,C 180,E1 -3237.812,E2 -3237.812} C_VEL
LIN {X 0,Y 552.241,Z 330.321,A -85,B 0,C 180,E1 -3240.729,E2 -3240.729} C_VEL
LIN {X 0,Y 552.205,Z 330.325,A -85,B 0,C 180,E1 -3242.918,E2 -3242.918} C_VEL
LIN {X 0,Y 552.193,Z 330.321,A -85,B 0,C 180,E1 -3245.844,E2 -3245.844} C_VEL
LIN {X 0,Y 552.163,Z 330.331,A -85,B 0,C 180,E1 -3248.786,E2 -3248.786} C_VEL
LIN {X 0,Y 552.155,Z 330.325,A -85,B 0,C 180,E1 -3251.751,E2 -3251.751} C_VEL
LIN {X 0,Y 552.126,Z 330.335,A -85,B 0,C 180,E1 -3254.749,E2 -3254.749} C_VEL
LIN {X 0,Y 552.107,Z 330.331,A -85,B 0,C 180,E1 -3257.789,E2 -3257.789} C_VEL
LIN {X 0,Y 552.125,Z 330.331,A -85,B 0,C 180,E1 -3260.101,E2 -3260.101} C_VEL
LIN {X 0,Y 552.106,Z 330.337,A -85,B 0,C 180,E1 -3262.45,E2 -3262.45} C_VEL
LIN {X 0,Y 552.147,Z 330.326,A -85,B 0,C 180,E1 -3265.351,E2 -3265.351} C_VEL
LIN {X 0,Y 552.118,Z 330.328,A -85,B 0,C 180,E1 -3268.098,E2 -3268.098} C_VEL
LIN {X 0,Y 552.099,Z 330.337,A -85,B 0,C 180,E1 -3270.609,E2 -3270.609} C_VEL
LIN {X 0,Y 552.121,Z 330.331,A -85,B 0,C 180,E1 -3273.185,E2 -3273.185} C_VEL
LIN {X 0,Y 552.105,Z 330.334,A -85,B 0,C 180,E1 -3275.842,E2 -3275.842} C_VEL
LIN {X 0,Y 552.118,Z 330.328,A -85,B 0,C 180,E1 -3279.063,E2 -3279.063} C_VEL
LIN {X 0,Y 552.165,Z 330.325,A -85,B 0,C 180,E1 -3281.442,E2 -3281.442} C_VEL
LIN {X 0,Y 552.09,Z 330.334,A -85,B 0,C 180,E1 -3284.533,E2 -3284.533} C_VEL
LIN {X 0,Y 552.124,Z 330.332,A -85,B 0,C 180,E1 -3287.585,E2 -3287.585} C_VEL
LIN {X 0,Y 552.13,Z 330.332,A -85,B 0,C 180,E1 -3290.474,E2 -3290.474} C_VEL
LIN {X 0,Y 552.11,Z 330.333,A -85,B 0,C 180,E1 -3293.317,E2 -3293.317} C_VEL
LIN {X 0,Y 552.137,Z 330.338,A -85,B 0,C 180,E1 -3295.941,E2 -3295.941} C_VEL
LIN {X 0,Y 552.115,Z 330.334,A -85,B 0,C 180,E1 -3298.542,E2 -3298.542} C_VEL
LIN {X 0,Y 552.124,Z 330.326,A -85,B 0,C 180,E1 -3301.438,E2 -3301.438} C_VEL
LIN {X 0,Y 552.135,Z 330.328,A -85,B 0,C 180,E1 -3304.357,E2 -3304.357} C_VEL
LIN {X 0,Y 552.127,Z 330.522,A -85,B 0,C 180,E1 -3306.351,E2 -3306.351} C_VEL
LIN {X 0,Y 553.361,Z 337.02,A -85,B 0,C 180,E1 -3307.408,E2 -3307.408} C_VEL
LIN {X 0,Y 552.957,Z 357.315,A -85,B 0,C 180,E1 -3310.419,E2 -3310.419} C_VEL
LIN {X 0,Y 552.717,Z 372.236,A -85,B 0,C 180,E1 -3312.563,E2 -3312.563} C_VEL
LIN {X 0,Y 554.003,Z 379.219,A -85,B 0,C 180,E1 -3312.727,E2 -3312.727} C_VEL
LIN {X 0,Y 554.198,Z 391.53,A -85,B 0,C 180,E1 -3312.897,E2 -3312.897} C_VEL
LIN {X 0,Y 553.777,Z 508.697,A -85,B 0,C 180,E1 -3314.45,E2 -3314.45} C_VEL
LIN {X 0,Y 553.579,Z 523.198,A -85,B 0,C 180,E1 -3314.784,E2 -3314.784} C_VEL
LIN {X 0,Y 553.374,Z 537.721,A -85,B 0,C 180,E1 -3315.286,E2 -3315.286} C_VEL
LIN {X 0,Y 553.166,Z 551.659,A -85,B 0,C 180,E1 -3315.938,E2 -3315.938} C_VEL
LIN {X 0,Y 552.895,Z 564.118,A -85,B 0,C 180,E1 -3316.681,E2 -3316.681} C_VEL
LIN {X 0,Y 552.629,Z 576.659,A -85,B 0,C 180,E1 -3317.609,E2 -3317.609} C_VEL
LIN {X 0,Y 552.445,Z 587.304,A -85,B 0,C 180,E1 -3318.573,E2 -3318.573} C_VEL
LIN {X 0,Y 552.178,Z 597.861,A -85,B 0,C 180,E1 -3319.737,E2 -3319.737} C_VEL
LIN {X 0,Y 552.031,Z 606.181,A -85,B 0,C 180,E1 -3320.844,E2 -3320.844} C_VEL
LIN {X 0,Y 551.912,Z 614.133,A -85,B 0,C 180,E1 -3322.133,E2 -3322.133} C_VEL
LIN {X 0,Y 551.821,Z 620.531,A -85,B 0,C 180,E1 -3323.419,E2 -3323.419} C_VEL
LIN {X 0,Y 551.792,Z 624.963,A -85,B 0,C 180,E1 -3324.519,E2 -3324.519} C_VEL
LIN {X 0,Y 551.759,Z 628.449,A -85,B 0,C 180,E1 -3325.618,E2 -3325.618} C_VEL
LIN {X 0,Y 551.72,Z 631.837,A -85,B 0,C 180,E1 -3327.08,E2 -3327.08} C_VEL
LIN {X 0,Y 551.64,Z 633.836,A -85,B 0,C 180,E1 -3328.541,E2 -3328.541} C_VEL
LIN {X 0,Y 551.639,Z 634.5,A -85,B 0,C 180,E1 -3330.001,E2 -3330.001} C_VEL
LIN {X 0,Y 551.64,Z 633.833,A -85,B 0,C 180,E1 -3331.461,E2 -3331.461} C_VEL
LIN {X 0,Y 551.72,Z 631.83,A -85,B 0,C 180,E1 -3332.922,E2 -3332.922} C_VEL
LIN {X 0,Y 551.76,Z 628.441,A -85,B 0,C 180,E1 -3334.384,E2 -3334.384} C_VEL
LIN {X 0,Y 551.825,Z 623.565,A -85,B 0,C 180,E1 -3335.849,E2 -3335.849} C_VEL
LIN {X 0,Y 551.834,Z 617.05,A -85,B 0,C 180,E1 -3337.318,E2 -3337.318} C_VEL
LIN {X 0,Y 551.963,Z 609.797,A -85,B 0,C 180,E1 -3338.605,E2 -3338.605} C_VEL
LIN {X 0,Y 552.116,Z 600.815,A -85,B 0,C 180,E1 -3339.896,E2 -3339.896} C_VEL
LIN {X 0,Y 552.347,Z 591.384,A -85,B 0,C 180,E1 -3341.004,E2 -3341.004} C_VEL
LIN {X 0,Y 552.54,Z 580.945,A -85,B 0,C 180,E1 -3342.022,E2 -3342.022} C_VEL
LIN {X 0,Y 552.762,Z 569.417,A -85,B 0,C 180,E1 -3342.95,E2 -3342.95} C_VEL
LIN {X 0,Y 553.013,Z 556.623,A -85,B 0,C 180,E1 -3343.786,E2 -3343.786} C_VEL
LIN {X 0,Y 553.285,Z 544.134,A -85,B 0,C 180,E1 -3344.436,E2 -3344.436} C_VEL
LIN {X 0,Y 553.532,Z 531.055,A -85,B 0,C 180,E1 -3344.964,E2 -3344.964} C_VEL
LIN {X 0,Y 553.673,Z 517.424,A -85,B 0,C 180,E1 -3345.366,E2 -3345.366} C_VEL
LIN {X 0,Y 553.783,Z 502.544,A -85,B 0,C 180,E1 -3345.646,E2 -3345.646} C_VEL
LIN {X 0,Y 554.133,Z 379.965,A -85,B 0,C 180,E1 -3347.259,E2 -3347.259} C_VEL
LIN {X 0,Y 552.753,Z 372.402,A -85,B 0,C 180,E1 -3347.425,E2 -3347.425} C_VEL
LIN {X 0,Y 552.795,Z 364.467,A -85,B 0,C 180,E1 -3348.533,E2 -3348.533} C_VEL
LIN {X 0,Y 553.144,Z 346.16,A -85,B 0,C 180,E1 -3351.231,E2 -3351.231} C_VEL
LIN {X 0,Y 553.326,Z 337.007,A -85,B 0,C 180,E1 -3352.596,E2 -3352.596} C_VEL
LIN {X 0,Y 552.129,Z 330.456,A -85,B 0,C 180,E1 -3353.667,E2 -3353.667} C_VEL
LIN {X 0,Y 552.125,Z 330.337,A -85,B 0,C 180,E1 -3356.457,E2 -3356.457} C_VEL
LIN {X 0,Y 552.116,Z 330.328,A -85,B 0,C 180,E1 -3358.929,E2 -3358.929} C_VEL
LIN {X 0,Y 552.115,Z 330.333,A -85,B 0,C 180,E1 -3361.476,E2 -3361.476} C_VEL
LIN {X 0,Y 552.144,Z 330.335,A -85,B 0,C 180,E1 -3364.172,E2 -3364.172} C_VEL
LIN {X 0,Y 552.117,Z 330.333,A -85,B 0,C 180,E1 -3366.747,E2 -3366.747} C_VEL
LIN {X 0,Y 552.135,Z 330.333,A -85,B 0,C 180,E1 -3369.528,E2 -3369.528} C_VEL
LIN {X 0,Y 552.134,Z 330.331,A -85,B 0,C 180,E1 -3372.426,E2 -3372.426} C_VEL
LIN {X 0,Y 552.102,Z 330.338,A -85,B 0,C 180,E1 -3375.563,E2 -3375.563} C_VEL
LIN {X 0,Y 552.135,Z 330.33,A -85,B 0,C 180,E1 -3378.555,E2 -3378.555} C_VEL
LIN {X 0,Y 552.121,Z 330.335,A -85,B 0,C 180,E1 -3381.411,E2 -3381.411} C_VEL
LIN {X 0,Y 552.089,Z 330.338,A -85,B 0,C 180,E1 -3384.157,E2 -3384.157} C_VEL
LIN {X 0,Y 552.12,Z 330.332,A -85,B 0,C 180,E1 -3386.814,E2 -3386.814} C_VEL
LIN {X 0,Y 552.107,Z 330.34,A -85,B 0,C 180,E1 -3389.391,E2 -3389.391} C_VEL
LIN {X 0,Y 552.125,Z 330.338,A -85,B 0,C 180,E1 -3391.903,E2 -3391.903} C_VEL
LIN {X 0,Y 552.182,Z 330.481,A -85,B 0,C 180,E1 -3394.257,E2 -3394.257} C_VEL
LIN {X 0,Y 553.435,Z 338.027,A -85,B 0,C 180,E1 -3395.225,E2 -3395.225} C_VEL
LIN {X 0,Y 553.306,Z 355.403,A -85,B 0,C 180,E1 -3397.404,E2 -3397.404} C_VEL
LIN {X 0,Y 553.11,Z 375.999,A -85,B 0,C 180,E1 -3399.936,E2 -3399.936} C_VEL
LIN {X 0,Y 552.819,Z 398.063,A -85,B 0,C 180,E1 -3402.721,E2 -3402.721} C_VEL
LIN {X 0,Y 552.572,Z 421.385,A -85,B 0,C 180,E1 -3405.652,E2 -3405.652} C_VEL
LIN {X 0,Y 553.444,Z 428.156,A -85,B 0,C 180,E1 -3405.78,E2 -3405.78} C_VEL
LIN {X 0,Y 553.142,Z 530.439,A -85,B 0,C 180,E1 -3407.13,E2 -3407.13} C_VEL
LIN {X 0,Y 553.011,Z 543.843,A -85,B 0,C 180,E1 -3407.453,E2 -3407.453} C_VEL
LIN {X 0,Y 552.854,Z 555.908,A -85,B 0,C 180,E1 -3407.892,E2 -3407.892} C_VEL
LIN {X 0,Y 552.683,Z 568.44,A -85,B 0,C 180,E1 -3408.51,E2 -3408.51} C_VEL
LIN {X 0,Y 552.484,Z 579.108,A -85,B 0,C 180,E1 -3409.185,E2 -3409.185} C_VEL
LIN {X 0,Y 552.267,Z 589.588,A -85,B 0,C 180,E1 -3410.015,E2 -3410.015} C_VEL
LIN {X 0,Y 552.127,Z 599.902,A -85,B 0,C 180,E1 -3411.029,E2 -3411.029} C_VEL
LIN {X 0,Y 551.961,Z 608.86,A -85,B 0,C 180,E1 -3412.133,E2 -3412.133} C_VEL
LIN {X 0,Y 551.873,Z 615.191,A -85,B 0,C 180,E1 -3413.088,E2 -3413.088} C_VEL
LIN {X 0,Y 551.868,Z 620.959,A -85,B 0,C 180,E1 -3414.153,E2 -3414.153} C_VEL
LIN {X 0,Y 551.725,Z 625.697,A -85,B 0,C 180,E1 -3415.251,E2 -3415.251} C_VEL
LIN {X 0,Y 551.751,Z 629.326,A -85,B 0,C 180,E1 -3416.349,E2 -3416.349} C_VEL
LIN {X 0,Y 551.724,Z 631.196,A -85,B 0,C 180,E1 -3417.079,E2 -3417.079} C_VEL
LIN {X 0,Y 551.656,Z 632.63,A -85,B 0,C 180,E1 -3417.81,E2 -3417.81} C_VEL
LIN {X 0,Y 551.642,Z 634.256,A -85,B 0,C 180,E1 -3419.27,E2 -3419.27} C_VEL
LIN {X 0,Y 551.641,Z 634.496,A -85,B 0,C 180,E1 -3420,E2 -3420} C_VEL
LIN {X 0,Y 551.642,Z 634.313,A -85,B 0,C 180,E1 -3420.73,E2 -3420.73} C_VEL
LIN {X 0,Y 551.655,Z 632.767,A -85,B 0,C 180,E1 -3422.19,E2 -3422.19} C_VEL
LIN {X 0,Y 551.724,Z 631.406,A -85,B 0,C 180,E1 -3422.921,E2 -3422.921} C_VEL
LIN {X 0,Y 551.764,Z 628.535,A -85,B 0,C 180,E1 -3424.017,E2 -3424.017} C_VEL
LIN {X 0,Y 551.724,Z 624.636,A -85,B 0,C 180,E1 -3425.116,E2 -3425.116} C_VEL
LIN {X 0,Y 551.81,Z 618.887,A -85,B 0,C 180,E1 -3426.348,E2 -3426.348} C_VEL
LIN {X 0,Y 551.928,Z 612.046,A -85,B 0,C 180,E1 -3427.5,E2 -3427.5} C_VEL
LIN {X 0,Y 552.063,Z 603.871,A -85,B 0,C 180,E1 -3428.603,E2 -3428.603} C_VEL
LIN {X 0,Y 552.196,Z 595.464,A -85,B 0,C 180,E1 -3429.524,E2 -3429.524} C_VEL
LIN {X 0,Y 552.392,Z 585.161,A -85,B 0,C 180,E1 -3430.446,E2 -3430.446} C_VEL
LIN {X 0,Y 552.585,Z 574.363,A -85,B 0,C 180,E1 -3431.224,E2 -3431.224} C_VEL
LIN {X 0,Y 552.745,Z 563.772,A -85,B 0,C 180,E1 -3431.831,E2 -3431.831} C_VEL
LIN {X 0,Y 552.941,Z 551.182,A -85,B 0,C 180,E1 -3432.385,E2 -3432.385} C_VEL
LIN {X 0,Y 553.033,Z 538.786,A -85,B 0,C 180,E1 -3432.78,E2 -3432.78} C_VEL
LIN {X 0,Y 553.175,Z 526.063,A -85,B 0,C 180,E1 -3433.033,E2 -3433.033} C_VEL
LIN {X 0,Y 553.301,Z 426.959,A -85,B 0,C 180,E1 -3434.329,E2 -3434.329} C_VEL
LIN {X 0,Y 552.544,Z 421.315,A -85,B 0,C 180,E1 -3434.443,E2 -3434.443} C_VEL
LIN {X 0,Y 552.831,Z 396.656,A -85,B 0,C 180,E1 -3437.548,E2 -3437.548} C_VEL
LIN {X 0,Y 552.844,Z 396.03,A -85,B 0,C 180,E1 -3437.627,E2 -3437.627} C_VEL
LIN {X 0,Y 552.261,Z 392.402,A -85,B 0,C 180,E1 -3438.107,E2 -3438.107} C_VEL
LIN {X 0,Y 546.791,Z 381.197,A -85,B 0,C 180,E1 -3439.719,E2 -3439.719} C_VEL
LIN {X 0,Y 546.204,Z 377.567,A -85,B 0,C 180,E1 -3440.207,E2 -3440.207} C_VEL
LIN {X 0,Y 546.613,Z 355.156,A -85,B 0,C 180,E1 -3443.088,E2 -3443.088} C_VEL
LIN {X 0,Y 546.74,Z 339.632,A -85,B 0,C 180,E1 -3445.1,E2 -3445.1} C_VEL
LIN {X 0,Y 545.112,Z 331.336,A -85,B 0,C 180,E1 -3446.282,E2 -3446.282} C_VEL
LIN {X 0,Y 545.07,Z 331.212,A -85,B 0,C 180,E1 -3449.338,E2 -3449.338} C_VEL
LIN {X 0,Y 545.061,Z 331.214,A -85,B 0,C 180,E1 -3451.915,E2 -3451.915} C_VEL
LIN {X 0,Y 545.067,Z 331.216,A -85,B 0,C 180,E1 -3454.564,E2 -3454.564} C_VEL
LIN {X 0,Y 545.041,Z 331.213,A -85,B 0,C 180,E1 -3457.304,E2 -3457.304} C_VEL
LIN {X 0,Y 545.07,Z 331.216,A -85,B 0,C 180,E1 -3460.142,E2 -3460.142} C_VEL
LIN {X 0,Y 545.084,Z 331.206,A -85,B 0,C 180,E1 -3463.106,E2 -3463.106} C_VEL
LIN {X 0,Y 545.072,Z 331.214,A -85,B 0,C 180,E1 -3466.224,E2 -3466.224} C_VEL
LIN {X 0,Y 545.086,Z 331.206,A -85,B 0,C 180,E1 -3468.885,E2 -3468.885} C_VEL
LIN {X 0,Y 545.086,Z 331.206,A -85,B 0,C 180,E1 -3470.818,E2 -3470.818} C_VEL
LIN {X 0,Y 545.055,Z 331.214,A -85,B 0,C 180,E1 -3473.62,E2 -3473.62} C_VEL
LIN {X 0,Y 545.073,Z 331.212,A -85,B 0,C 180,E1 -3476.328,E2 -3476.328} C_VEL
LIN {X 0,Y 545.072,Z 331.21,A -85,B 0,C 180,E1 -3478.952,E2 -3478.952} C_VEL
LIN {X 0,Y 545.108,Z 331.199,A -85,B 0,C 180,E1 -3481.507,E2 -3481.507} C_VEL
LIN {X 0,Y 545.101,Z 331.204,A -85,B 0,C 180,E1 -3484.491,E2 -3484.491} C_VEL
LIN {X 0,Y 545.126,Z 331.434,A -85,B 0,C 180,E1 -3486.214,E2 -3486.214} C_VEL
LIN {X 0,Y 546.403,Z 338.02,A -85,B 0,C 180,E1 -3487.302,E2 -3487.302} C_VEL
LIN {X 0,Y 546.031,Z 356.617,A -85,B 0,C 180,E1 -3490.101,E2 -3490.101} C_VEL
LIN {X 0,Y 545.74,Z 371.982,A -85,B 0,C 180,E1 -3492.358,E2 -3492.358} C_VEL
LIN {X 0,Y 546.108,Z 374.409,A -85,B 0,C 180,E1 -3492.449,E2 -3492.449} C_VEL
LIN {X 0,Y 547.479,Z 382.584,A -85,B 0,C 180,E1 -3492.605,E2 -3492.605} C_VEL
LIN {X 0,Y 546.925,Z 508.23,A -85,B 0,C 180,E1 -3494.296,E2 -3494.296} C_VEL
LIN {X 0,Y 546.79,Z 519.496,A -85,B 0,C 180,E1 -3494.541,E2 -3494.541} C_VEL
LIN {X 0,Y 546.676,Z 528.18,A -85,B 0,C 180,E1 -3494.795,E2 -3494.795} C_VEL
LIN {X 0,Y 546.463,Z 538.773,A -85,B 0,C 180,E1 -3495.189,E2 -3495.189} C_VEL
LIN {X 0,Y 546.283,Z 550.663,A -85,B 0,C 180,E1 -3495.756,E2 -3495.756} C_VEL
LIN {X 0,Y 545.996,Z 560.412,A -85,B 0,C 180,E1 -3496.318,E2 -3496.318} C_VEL
LIN {X 0,Y 545.792,Z 569.994,A -85,B 0,C 180,E1 -3496.976,E2 -3496.976} C_VEL
LIN {X 0,Y 545.548,Z 579.286,A -85,B 0,C 180,E1 -3497.727,E2 -3497.727} C_VEL
LIN {X 0,Y 545.396,Z 587.389,A -85,B 0,C 180,E1 -3498.488,E2 -3498.488} C_VEL
LIN {X 0,Y 545.224,Z 595.854,A -85,B 0,C 180,E1 -3499.415,E2 -3499.415} C_VEL
LIN {X 0,Y 545.026,Z 603.169,A -85,B 0,C 180,E1 -3500.349,E2 -3500.349} C_VEL
LIN {X 0,Y 544.911,Z 609.454,A -85,B 0,C 180,E1 -3501.283,E2 -3501.283} C_VEL
LIN {X 0,Y 544.826,Z 614.869,A -85,B 0,C 180,E1 -3502.215,E2 -3502.215} C_VEL
LIN {X 0,Y 544.736,Z 620.715,A -85,B 0,C 180,E1 -3503.429,E2 -3503.429} C_VEL
LIN {X 0,Y 544.724,Z 624.747,A -85,B 0,C 180,E1 -3504.446,E2 -3504.446} C_VEL
LIN {X 0,Y 544.655,Z 628.299,A -85,B 0,C 180,E1 -3505.559,E2 -3505.559} C_VEL
LIN {X 0,Y 544.658,Z 630.216,A -85,B 0,C 180,E1 -3506.3,E2 -3506.3} C_VEL
LIN {X 0,Y 544.57,Z 632.94,A -85,B 0,C 180,E1 -3507.78,E2 -3507.78} C_VEL
LIN {X 0,Y 544.537,Z 634.252,A -85,B 0,C 180,E1 -3509.26,E2 -3509.26} C_VEL
LIN {X 0,Y 544.54,Z 634.496,A -85,B 0,C 180,E1 -3509.999,E2 -3509.999} C_VEL
LIN {X 0,Y 544.542,Z 633.847,A -85,B 0,C 180,E1 -3511.478,E2 -3511.478} C_VEL
LIN {X 0,Y 544.645,Z 631.86,A -85,B 0,C 180,E1 -3512.958,E2 -3512.958} C_VEL
LIN {X 0,Y 544.658,Z 630.436,A -85,B 0,C 180,E1 -3513.698,E2 -3513.698} C_VEL
LIN {X 0,Y 544.646,Z 626.313,A -85,B 0,C 180,E1 -3515.181,E2 -3515.181} C_VEL
LIN {X 0,Y 544.691,Z 622.199,A -85,B 0,C 180,E1 -3516.309,E2 -3516.309} C_VEL
LIN {X 0,Y 544.78,Z 617.238,A -85,B 0,C 180,E1 -3517.411,E2 -3517.411} C_VEL
LIN {X 0,Y 544.895,Z 611.141,A -85,B 0,C 180,E1 -3518.529,E2 -3518.529} C_VEL
LIN {X 0,Y 545.016,Z 605.153,A -85,B 0,C 180,E1 -3519.462,E2 -3519.462} C_VEL
LIN {X 0,Y 545.15,Z 598.17,A -85,B 0,C 180,E1 -3520.397,E2 -3520.397} C_VEL
LIN {X 0,Y 545.335,Z 590.105,A -85,B 0,C 180,E1 -3521.321,E2 -3521.321} C_VEL
LIN {X 0,Y 545.518,Z 581.37,A -85,B 0,C 180,E1 -3522.178,E2 -3522.178} C_VEL
LIN {X 0,Y 545.726,Z 572.431,A -85,B 0,C 180,E1 -3522.929,E2 -3522.929} C_VEL
LIN {X 0,Y 545.939,Z 563.289,A -85,B 0,C 180,E1 -3523.587,E2 -3523.587} C_VEL
LIN {X 0,Y 546.199,Z 552.355,A -85,B 0,C 180,E1 -3524.245,E2 -3524.245} C_VEL
LIN {X 0,Y 546.392,Z 541.913,A -85,B 0,C 180,E1 -3524.763,E2 -3524.763} C_VEL
LIN {X 0,Y 546.642,Z 531.14,A -85,B 0,C 180,E1 -3525.192,E2 -3525.192} C_VEL
LIN {X 0,Y 546.774,Z 520.277,A -85,B 0,C 180,E1 -3525.529,E2 -3525.529} C_VEL
LIN {X 0,Y 546.9,Z 509.378,A -85,B 0,C 180,E1 -3525.775,E2 -3525.775} C_VEL
LIN {X 0,Y 547.1,Z 475.648,A -85,B 0,C 180,E1 -3526.247,E2 -3526.247} C_VEL
LIN {X 0,Y 547.323,Z 380.652,A -85,B 0,C 180,E1 -3527.516,E2 -3527.516} C_VEL
LIN {X 0,Y 545.764,Z 372.42,A -85,B 0,C 180,E1 -3527.698,E2 -3527.698} C_VEL
LIN {X 0,Y 545.805,Z 368.706,A -85,B 0,C 180,E1 -3528.194,E2 -3528.194} C_VEL
LIN {X 0,Y 546.168,Z 350.395,A -85,B 0,C 180,E1 -3530.92,E2 -3530.92} C_VEL
LIN {X 0,Y 546.453,Z 338.622,A -85,B 0,C 180,E1 -3532.694,E2 -3532.694} C_VEL
LIN {X 0,Y 545.095,Z 331.278,A -85,B 0,C 180,E1 -3533.924,E2 -3533.924} C_VEL
LIN {X 0,Y 545.104,Z 331.209,A -85,B 0,C 180,E1 -3536.823,E2 -3536.823} C_VEL
LIN {X 0,Y 545.081,Z 331.199,A -85,B 0,C 180,E1 -3539.336,E2 -3539.336} C_VEL
LIN {X 0,Y 545.07,Z 331.216,A -85,B 0,C 180,E1 -3541.912,E2 -3541.912} C_VEL
LIN {X 0,Y 545.082,Z 331.21,A -85,B 0,C 180,E1 -3544.562,E2 -3544.562} C_VEL
LIN {X 0,Y 545.036,Z 331.214,A -85,B 0,C 180,E1 -3547.302,E2 -3547.302} C_VEL
LIN {X 0,Y 545.089,Z 331.211,A -85,B 0,C 180,E1 -3550.139,E2 -3550.139} C_VEL
LIN {X 0,Y 545.081,Z 331.208,A -85,B 0,C 180,E1 -3553.105,E2 -3553.105} C_VEL
LIN {X 0,Y 545.061,Z 331.212,A -85,B 0,C 180,E1 -3556.223,E2 -3556.223} C_VEL
LIN {X 0,Y 545.117,Z 331.203,A -85,B 0,C 180,E1 -3558.888,E2 -3558.888} C_VEL
LIN {X 0,Y 545.047,Z 331.211,A -85,B 0,C 180,E1 -3561.762,E2 -3561.762} C_VEL
LIN {X 0,Y 545.056,Z 331.209,A -85,B 0,C 180,E1 -3564.533,E2 -3564.533} C_VEL
LIN {X 0,Y 545.075,Z 331.212,A -85,B 0,C 180,E1 -3567.212,E2 -3567.212} C_VEL
LIN {X 0,Y 545.093,Z 331.201,A -85,B 0,C 180,E1 -3569.812,E2 -3569.812} C_VEL
LIN {X 0,Y 545.093,Z 331.2,A -85,B 0,C 180,E1 -3572.824,E2 -3572.824} C_VEL
LIN {X 0,Y 545.051,Z 331.218,A -85,B 0,C 180,E1 -3575.631,E2 -3575.631} C_VEL
LIN {X 0,Y 545.071,Z 331.206,A -85,B 0,C 180,E1 -3578.175,E2 -3578.175} C_VEL
LIN {X 0,Y 545.111,Z 331.203,A -85,B 0,C 180,E1 -3580.414,E2 -3580.414} C_VEL
LIN {X 0,Y 545.07,Z 331.211,A -85,B 0,C 180,E1 -3583.521,E2 -3583.521} C_VEL
LIN {X 0,Y 545.086,Z 331.208,A -85,B 0,C 180,E1 -3585.82,E2 -3585.82} C_VEL
LIN {X 0,Y 545.135,Z 331.203,A -85,B 0,C 180,E1 -3588.85,E2 -3588.85} C_VEL
LIN {X 0,Y 545.127,Z 331.201,A -85,B 0,C 180,E1 -3591.847,E2 -3591.847} C_VEL
LIN {X 0,Y 545.201,Z 331.197,A -85,B 0,C 180,E1 -3594.823,E2 -3594.823} C_VEL
LIN {X 0,Y 545.187,Z 331.193,A -85,B 0,C 180,E1 -3597.784,E2 -3597.784} C_VEL
LIN {X 0,Y 545.21,Z 331.197,A -85,B 0,C 180,E1 -3600.739,E2 -3600.739} C_VEL
LIN {X 0,Y 545.17,Z 331.201,A -85,B 0,C 180,E1 -3602.956,E2 -3602.956} C_VEL
LIN {X 0,Y 545.164,Z 331.196,A -85,B 0,C 180,E1 -3605.92,E2 -3605.92} C_VEL
LIN {X 0,Y 545.12,Z 331.206,A -85,B 0,C 180,E1 -3608.9,E2 -3608.9} C_VEL
LIN {X 0,Y 545.126,Z 331.201,A -85,B 0,C 180,E1 -3611.904,E2 -3611.904} C_VEL
LIN {X 0,Y 545.076,Z 331.21,A -85,B 0,C 180,E1 -3614.944,E2 -3614.944} C_VEL
LIN {X 0,Y 545.075,Z 331.208,A -85,B 0,C 180,E1 -3618.026,E2 -3618.026} C_VEL
LIN {X 0,Y 545.09,Z 331.21,A -85,B 0,C 180,E1 -3620.372,E2 -3620.372} C_VEL
LIN {X 0,Y 545.105,Z 331.204,A -85,B 0,C 180,E1 -3623.558,E2 -3623.558} C_VEL
LIN {X 0,Y 545.08,Z 331.208,A -85,B 0,C 180,E1 -3626.001,E2 -3626.001} C_VEL
LIN {X 0,Y 545.082,Z 331.201,A -85,B 0,C 180,E1 -3628.749,E2 -3628.749} C_VEL
LIN {X 0,Y 545.069,Z 331.207,A -85,B 0,C 180,E1 -3631.683,E2 -3631.683} C_VEL
LIN {X 0,Y 545.076,Z 331.213,A -85,B 0,C 180,E1 -3634.564,E2 -3634.564} C_VEL
LIN {X 0,Y 545.031,Z 331.206,A -85,B 0,C 180,E1 -3637.304,E2 -3637.304} C_VEL
LIN {X 0,Y 545.086,Z 331.211,A -85,B 0,C 180,E1 -3640.141,E2 -3640.141} C_VEL
LIN {X 0,Y 545.061,Z 331.211,A -85,B 0,C 180,E1 -3642.698,E2 -3642.698} C_VEL
LIN {X 0,Y 545.056,Z 331.205,A -85,B 0,C 180,E1 -3645.168,E2 -3645.168} C_VEL
LIN {X 0,Y 545.077,Z 331.214,A -85,B 0,C 180,E1 -3647.899,E2 -3647.899} C_VEL
LIN {X 0,Y 545.101,Z 331.205,A -85,B 0,C 180,E1 -3650.677,E2 -3650.677} C_VEL
LIN {X 0,Y 545.052,Z 331.215,A -85,B 0,C 180,E1 -3653.622,E2 -3653.622} C_VEL
LIN {X 0,Y 545.075,Z 331.211,A -85,B 0,C 180,E1 -3656.33,E2 -3656.33} C_VEL
LIN {X 0,Y 545.067,Z 331.21,A -85,B 0,C 180,E1 -3658.954,E2 -3658.954} C_VEL
LIN {X 0,Y 545.102,Z 331.201,A -85,B 0,C 180,E1 -3661.509,E2 -3661.509} C_VEL
LIN {X 0,Y 545.097,Z 331.204,A -85,B 0,C 180,E1 -3664.491,E2 -3664.491} C_VEL
LIN {X 0,Y 545.106,Z 331.434,A -85,B 0,C 180,E1 -3666.172,E2 -3666.172} C_VEL
LIN {X 0,Y 546.44,Z 338.328,A -85,B 0,C 180,E1 -3667.305,E2 -3667.305} C_VEL
LIN {X 0,Y 546.024,Z 358.089,A -85,B 0,C 180,E1 -3670.276,E2 -3670.276} C_VEL
LIN {X 0,Y 545.765,Z 372.146,A -85,B 0,C 180,E1 -3672.329,E2 -3672.329} C_VEL
LIN {X 0,Y 546.782,Z 377.797,A -85,B 0,C 180,E1 -3672.473,E2 -3672.473} C_VEL
LIN {X 0,Y 547.42,Z 382.697,A -85,B 0,C 180,E1 -3672.56,E2 -3672.56} C_VEL
LIN {X 0,Y 546.938,Z 508.696,A -85,B 0,C 180,E1 -3674.251,E2 -3674.251} C_VEL
LIN {X 0,Y 546.773,Z 522.658,A -85,B 0,C 180,E1 -3674.573,E2 -3674.573} C_VEL
LIN {X 0,Y 546.557,Z 536.714,A -85,B 0,C 180,E1 -3675.056,E2 -3675.056} C_VEL
LIN {X 0,Y 546.314,Z 549.891,A -85,B 0,C 180,E1 -3675.663,E2 -3675.663} C_VEL
LIN {X 0,Y 545.966,Z 562.691,A -85,B 0,C 180,E1 -3676.414,E2 -3676.414} C_VEL
LIN {X 0,Y 545.707,Z 574.319,A -85,B 0,C 180,E1 -3677.26,E2 -3677.26} C_VEL
LIN {X 0,Y 545.448,Z 585.128,A -85,B 0,C 180,E1 -3678.213,E2 -3678.213} C_VEL
LIN {X 0,Y 545.231,Z 594.715,A -85,B 0,C 180,E1 -3679.229,E2 -3679.229} C_VEL
LIN {X 0,Y 545.025,Z 603.563,A -85,B 0,C 180,E1 -3680.351,E2 -3680.351} C_VEL
LIN {X 0,Y 544.872,Z 612.041,A -85,B 0,C 180,E1 -3681.658,E2 -3681.658} C_VEL
LIN {X 0,Y 544.735,Z 618.867,A -85,B 0,C 180,E1 -3682.961,E2 -3682.961} C_VEL
LIN {X 0,Y 544.73,Z 623.571,A -85,B 0,C 180,E1 -3684.077,E2 -3684.077} C_VEL
LIN {X 0,Y 544.654,Z 628.45,A -85,B 0,C 180,E1 -3685.561,E2 -3685.561} C_VEL
LIN {X 0,Y 544.646,Z 631.837,A -85,B 0,C 180,E1 -3687.042,E2 -3687.042} C_VEL
LIN {X 0,Y 544.541,Z 633.837,A -85,B 0,C 180,E1 -3688.522,E2 -3688.522} C_VEL
LIN {X 0,Y 544.539,Z 634.5,A -85,B 0,C 180,E1 -3690.001,E2 -3690.001} C_VEL
LIN {X 0,Y 544.541,Z 633.833,A -85,B 0,C 180,E1 -3691.48,E2 -3691.48} C_VEL
LIN {X 0,Y 544.647,Z 631.831,A -85,B 0,C 180,E1 -3692.96,E2 -3692.96} C_VEL
LIN {X 0,Y 544.654,Z 628.441,A -85,B 0,C 180,E1 -3694.441,E2 -3694.441} C_VEL
LIN {X 0,Y 544.735,Z 623.565,A -85,B 0,C 180,E1 -3695.925,E2 -3695.925} C_VEL
LIN {X 0,Y 544.784,Z 617.05,A -85,B 0,C 180,E1 -3697.413,E2 -3697.413} C_VEL
LIN {X 0,Y 544.911,Z 609.797,A -85,B 0,C 180,E1 -3698.717,E2 -3698.717} C_VEL
LIN {X 0,Y 545.082,Z 600.815,A -85,B 0,C 180,E1 -3700.025,E2 -3700.025} C_VEL
LIN {X 0,Y 545.333,Z 591.384,A -85,B 0,C 180,E1 -3701.147,E2 -3701.147} C_VEL
LIN {X 0,Y 545.546,Z 580.943,A -85,B 0,C 180,E1 -3702.179,E2 -3702.179} C_VEL
LIN {X 0,Y 545.797,Z 569.415,A -85,B 0,C 180,E1 -3703.118,E2 -3703.118} C_VEL
LIN {X 0,Y 546.119,Z 556.621,A -85,B 0,C 180,E1 -3703.964,E2 -3703.964} C_VEL
LIN {X 0,Y 546.41,Z 544.133,A -85,B 0,C 180,E1 -3704.622,E2 -3704.622} C_VEL
LIN {X 0,Y 546.677,Z 530.185,A -85,B 0,C 180,E1 -3705.188,E2 -3705.188} C_VEL
LIN {X 0,Y 546.887,Z 516.036,A -85,B 0,C 180,E1 -3705.598,E2 -3705.598} C_VEL
LIN {X 0,Y 546.971,Z 500.763,A -85,B 0,C 180,E1 -3705.87,E2 -3705.87} C_VEL
LIN {X 0,Y 547.435,Z 381.762,A -85,B 0,C 180,E1 -3707.452,E2 -3707.452} C_VEL
LIN {X 0,Y 545.774,Z 372.416,A -85,B 0,C 180,E1 -3707.653,E2 -3707.653} C_VEL
LIN {X 0,Y 545.808,Z 368.39,A -85,B 0,C 180,E1 -3708.196,E2 -3708.196} C_VEL
LIN {X 0,Y 546.178,Z 350.083,A -85,B 0,C 180,E1 -3710.922,E2 -3710.922} C_VEL
LIN {X 0,Y 546.414,Z 338.315,A -85,B 0,C 180,E1 -3712.698,E2 -3712.698} C_VEL
LIN {X 0,Y 545.091,Z 331.287,A -85,B 0,C 180,E1 -3713.875,E2 -3713.875} C_VEL
LIN {X 0,Y 545.085,Z 331.208,A -85,B 0,C 180,E1 -3716.001,E2 -3716.001} C_VEL
LIN {X 0,Y 545.095,Z 331.203,A -85,B 0,C 180,E1 -3718.749,E2 -3718.749} C_VEL
LIN {X 0,Y 545.062,Z 331.214,A -85,B 0,C 180,E1 -3721.679,E2 -3721.679} C_VEL
LIN {X 0,Y 545.087,Z 331.21,A -85,B 0,C 180,E1 -3724.563,E2 -3724.563} C_VEL
LIN {X 0,Y 545.044,Z 331.214,A -85,B 0,C 180,E1 -3727.304,E2 -3727.304} C_VEL
LIN {X 0,Y 545.071,Z 331.216,A -85,B 0,C 180,E1 -3730.143,E2 -3730.143} C_VEL
LIN {X 0,Y 545.083,Z 331.207,A -85,B 0,C 180,E1 -3733.107,E2 -3733.107} C_VEL
LIN {X 0,Y 545.072,Z 331.213,A -85,B 0,C 180,E1 -3736.225,E2 -3736.225} C_VEL
LIN {X 0,Y 545.091,Z 331.208,A -85,B 0,C 180,E1 -3738.886,E2 -3738.886} C_VEL
LIN {X 0,Y 545.057,Z 331.22,A -85,B 0,C 180,E1 -3741.763,E2 -3741.763} C_VEL
LIN {X 0,Y 545.04,Z 331.214,A -85,B 0,C 180,E1 -3744.532,E2 -3744.532} C_VEL
LIN {X 0,Y 545.074,Z 331.213,A -85,B 0,C 180,E1 -3747.212,E2 -3747.212} C_VEL
LIN {X 0,Y 545.068,Z 331.217,A -85,B 0,C 180,E1 -3749.811,E2 -3749.811} C_VEL
LIN {X 0,Y 545.094,Z 331.211,A -85,B 0,C 180,E1 -3752.344,E2 -3752.344} C_VEL
LIN {X 0,Y 545.154,Z 331.403,A -85,B 0,C 180,E1 -3754.144,E2 -3754.144} C_VEL
LIN {X 0,Y 546.424,Z 338.626,A -85,B 0,C 180,E1 -3755.088,E2 -3755.088} C_VEL
LIN {X 0,Y 546.457,Z 349.966,A -85,B 0,C 180,E1 -3756.504,E2 -3756.504} C_VEL
LIN {X 0,Y 546.179,Z 373.878,A -85,B 0,C 180,E1 -3759.473,E2 -3759.473} C_VEL
LIN {X 0,Y 545.939,Z 390.941,A -85,B 0,C 180,E1 -3761.615,E2 -3761.615} C_VEL
LIN {X 0,Y 545.622,Z 415.295,A -85,B 0,C 180,E1 -3764.728,E2 -3764.728} C_VEL
LIN {X 0,Y 545.568,Z 421.287,A -85,B 0,C 180,E1 -3765.459,E2 -3765.459} C_VEL
LIN {X 0,Y 546.569,Z 429.388,A -85,B 0,C 180,E1 -3765.615,E2 -3765.615} C_VEL
LIN {X 0,Y 546.244,Z 530.457,A -85,B 0,C 180,E1 -3766.964,E2 -3766.964} C_VEL
LIN {X 0,Y 546.086,Z 543.87,A -85,B 0,C 180,E1 -3767.291,E2 -3767.291} C_VEL
LIN {X 0,Y 545.901,Z 555.915,A -85,B 0,C 180,E1 -3767.736,E2 -3767.736} C_VEL
LIN {X 0,Y 545.736,Z 568.02,A -85,B 0,C 180,E1 -3768.338,E2 -3768.338} C_VEL
LIN {X 0,Y 545.499,Z 579.118,A -85,B 0,C 180,E1 -3769.045,E2 -3769.045} C_VEL
LIN {X 0,Y 545.261,Z 589.592,A -85,B 0,C 180,E1 -3769.886,E2 -3769.886} C_VEL
LIN {X 0,Y 545.102,Z 599.905,A -85,B 0,C 180,E1 -3770.913,E2 -3770.913} C_VEL
LIN {X 0,Y 544.918,Z 608.861,A -85,B 0,C 180,E1 -3772.031,E2 -3772.031} C_VEL
LIN {X 0,Y 544.797,Z 616.063,A -85,B 0,C 180,E1 -3773.147,E2 -3773.147} C_VEL
LIN {X 0,Y 544.778,Z 620.96,A -85,B 0,C 180,E1 -3774.076,E2 -3774.076} C_VEL
LIN {X 0,Y 544.629,Z 625.698,A -85,B 0,C 180,E1 -3775.189,E2 -3775.189} C_VEL
LIN {X 0,Y 544.67,Z 629.327,A -85,B 0,C 180,E1 -3776.301,E2 -3776.301} C_VEL
LIN {X 0,Y 544.651,Z 631.196,A -85,B 0,C 180,E1 -3777.041,E2 -3777.041} C_VEL
LIN {X 0,Y 544.571,Z 632.631,A -85,B 0,C 180,E1 -3777.781,E2 -3777.781} C_VEL
LIN {X 0,Y 544.542,Z 634.256,A -85,B 0,C 180,E1 -3779.261,E2 -3779.261} C_VEL
LIN {X 0,Y 544.541,Z 634.496,A -85,B 0,C 180,E1 -3780,E2 -3780} C_VEL
LIN {X 0,Y 544.542,Z 634.313,A -85,B 0,C 180,E1 -3780.74,E2 -3780.74} C_VEL
LIN {X 0,Y 544.57,Z 632.765,A -85,B 0,C 180,E1 -3782.219,E2 -3782.219} C_VEL
LIN {X 0,Y 544.651,Z 631.405,A -85,B 0,C 180,E1 -3782.959,E2 -3782.959} C_VEL
LIN {X 0,Y 544.684,Z 628.534,A -85,B 0,C 180,E1 -3784.07,E2 -3784.07} C_VEL
LIN {X 0,Y 544.653,Z 624.635,A -85,B 0,C 180,E1 -3785.182,E2 -3785.182} C_VEL
LIN {X 0,Y 544.723,Z 619.401,A -85,B 0,C 180,E1 -3786.333,E2 -3786.333} C_VEL
LIN {X 0,Y 544.861,Z 612.04,A -85,B 0,C 180,E1 -3787.597,E2 -3787.597} C_VEL
LIN {X 0,Y 545.016,Z 603.865,A -85,B 0,C 180,E1 -3788.715,E2 -3788.715} C_VEL
LIN {X 0,Y 545.158,Z 595.454,A -85,B 0,C 180,E1 -3789.648,E2 -3789.648} C_VEL
LIN {X 0,Y 545.357,Z 585.15,A -85,B 0,C 180,E1 -3790.582,E2 -3790.582} C_VEL
LIN {X 0,Y 545.599,Z 574.659,A -85,B 0,C 180,E1 -3791.35,E2 -3791.35} C_VEL
LIN {X 0,Y 545.787,Z 563.754,A -85,B 0,C 180,E1 -3791.984,E2 -3791.984} C_VEL
LIN {X 0,Y 546.01,Z 551.159,A -85,B 0,C 180,E1 -3792.545,E2 -3792.545} C_VEL
LIN {X 0,Y 546.132,Z 538.772,A -85,B 0,C 180,E1 -3792.944,E2 -3792.944} C_VEL
LIN {X 0,Y 546.266,Z 526.022,A -85,B 0,C 180,E1 -3793.201,E2 -3793.201} C_VEL
LIN {X 0,Y 546.443,Z 427.848,A -85,B 0,C 180,E1 -3794.499,E2 -3794.499} C_VEL
LIN {X 0,Y 545.538,Z 421.253,A -85,B 0,C 180,E1 -3794.635,E2 -3794.635} C_VEL
LIN {X 0,Y 545.83,Z 398.178,A -85,B 0,C 180,E1 -3797.553,E2 -3797.553} C_VEL
LIN {X 0,Y 546.204,Z 377.567,A -85,B 0,C 180,E1 -3800.207,E2 -3800.207} C_VEL
LIN {X 0,Y 545.611,Z 373.953,A -85,B 0,C 180,E1 -3800.693,E2 -3800.693} C_VEL
LIN {X 0,Y 540.155,Z 362.82,A -85,B 0,C 180,E1 -3802.333,E2 -3802.333} C_VEL
LIN {X 0,Y 539.597,Z 359.195,A -85,B 0,C 180,E1 -3802.827,E2 -3802.827} C_VEL
LIN {X 0,Y 539.878,Z 342.305,A -85,B 0,C 180,E1 -3805.029,E2 -3805.029} C_VEL
LIN {X 0,Y 538.468,Z 334.012,A -85,B 0,C 180,E1 -3806.182,E2 -3806.182} C_VEL
LIN {X 0,Y 538.078,Z 332.207,A -85,B 0,C 180,E1 -3806.469,E2 -3806.469} C_VEL
LIN {X 0,Y 538.036,Z 332.091,A -85,B 0,C 180,E1 -3808.933,E2 -3808.933} C_VEL
LIN {X 0,Y 538.016,Z 332.091,A -85,B 0,C 180,E1 -3811.887,E2 -3811.887} C_VEL
LIN {X 0,Y 538.017,Z 332.094,A -85,B 0,C 180,E1 -3814.617,E2 -3814.617} C_VEL
LIN {X 0,Y 538.009,Z 332.089,A -85,B 0,C 180,E1 -3817.17,E2 -3817.17} C_VEL
LIN {X 0,Y 538.027,Z 332.089,A -85,B 0,C 180,E1 -3819.797,E2 -3819.797} C_VEL
LIN {X 0,Y 538.024,Z 332.087,A -85,B 0,C 180,E1 -3822.786,E2 -3822.786} C_VEL
LIN {X 0,Y 538.033,Z 332.085,A -85,B 0,C 180,E1 -3825.925,E2 -3825.925} C_VEL
LIN {X 0,Y 538.053,Z 332.082,A -85,B 0,C 180,E1 -3829.252,E2 -3829.252} C_VEL
LIN {X 0,Y 537.998,Z 332.099,A -85,B 0,C 180,E1 -3832.122,E2 -3832.122} C_VEL
LIN {X 0,Y 538.018,Z 332.087,A -85,B 0,C 180,E1 -3834.916,E2 -3834.916} C_VEL
LIN {X 0,Y 538.024,Z 332.09,A -85,B 0,C 180,E1 -3837.617,E2 -3837.617} C_VEL
LIN {X 0,Y 538.023,Z 332.082,A -85,B 0,C 180,E1 -3840.238,E2 -3840.238} C_VEL
LIN {X 0,Y 538.069,Z 332.084,A -85,B 0,C 180,E1 -3842.796,E2 -3842.796} C_VEL
LIN {X 0,Y 538.034,Z 332.093,A -85,B 0,C 180,E1 -3845.703,E2 -3845.703} C_VEL
LIN {X 0,Y 538.073,Z 332.338,A -85,B 0,C 180,E1 -3846.022,E2 -3846.022} C_VEL
LIN {X 0,Y 539.472,Z 339.295,A -85,B 0,C 180,E1 -3847.19,E2 -3847.19} C_VEL
LIN {X 0,Y 539.15,Z 356.445,A -85,B 0,C 180,E1 -3849.809,E2 -3849.809} C_VEL
LIN {X 0,Y 538.785,Z 372.238,A -85,B 0,C 180,E1 -3852.145,E2 -3852.145} C_VEL
LIN {X 0,Y 540.283,Z 380.252,A -85,B 0,C 180,E1 -3852.333,E2 -3852.333} C_VEL
LIN {X 0,Y 540.702,Z 384.196,A -85,B 0,C 180,E1 -3852.401,E2 -3852.401} C_VEL
LIN {X 0,Y 540.095,Z 508.42,A -85,B 0,C 180,E1 -3854.092,E2 -3854.092} C_VEL
LIN {X 0,Y 539.942,Z 521.309,A -85,B 0,C 180,E1 -3854.385,E2 -3854.385} C_VEL
LIN {X 0,Y 539.779,Z 534.727,A -85,B 0,C 180,E1 -3854.828,E2 -3854.828} C_VEL
LIN {X 0,Y 539.496,Z 547.189,A -85,B 0,C 180,E1 -3855.38,E2 -3855.38} C_VEL
LIN {X 0,Y 539.146,Z 558.981,A -85,B 0,C 180,E1 -3856.044,E2 -3856.044} C_VEL
LIN {X 0,Y 538.838,Z 570.011,A -85,B 0,C 180,E1 -3856.805,E2 -3856.805} C_VEL
LIN {X 0,Y 538.592,Z 579.292,A -85,B 0,C 180,E1 -3857.566,E2 -3857.566} C_VEL
LIN {X 0,Y 538.37,Z 588.095,A -85,B 0,C 180,E1 -3858.411,E2 -3858.411} C_VEL
LIN {X 0,Y 538.209,Z 595.848,A -85,B 0,C 180,E1 -3859.275,E2 -3859.275} C_VEL
LIN {X 0,Y 537.978,Z 603.164,A -85,B 0,C 180,E1 -3860.221,E2 -3860.221} C_VEL
LIN {X 0,Y 537.864,Z 609.45,A -85,B 0,C 180,E1 -3861.168,E2 -3861.168} C_VEL
LIN {X 0,Y 537.771,Z 614.863,A -85,B 0,C 180,E1 -3862.112,E2 -3862.112} C_VEL
LIN {X 0,Y 537.668,Z 620.297,A -85,B 0,C 180,E1 -3863.243,E2 -3863.243} C_VEL
LIN {X 0,Y 537.656,Z 624.742,A -85,B 0,C 180,E1 -3864.373,E2 -3864.373} C_VEL
LIN {X 0,Y 537.55,Z 628.292,A -85,B 0,C 180,E1 -3865.5,E2 -3865.5} C_VEL
LIN {X 0,Y 537.577,Z 630.214,A -85,B 0,C 180,E1 -3866.251,E2 -3866.251} C_VEL
LIN {X 0,Y 537.489,Z 632.935,A -85,B 0,C 180,E1 -3867.751,E2 -3867.751} C_VEL
LIN {X 0,Y 537.438,Z 634.244,A -85,B 0,C 180,E1 -3869.25,E2 -3869.25} C_VEL
LIN {X 0,Y 537.441,Z 634.496,A -85,B 0,C 180,E1 -3869.999,E2 -3869.999} C_VEL
LIN {X 0,Y 537.447,Z 633.841,A -85,B 0,C 180,E1 -3871.498,E2 -3871.498} C_VEL
LIN {X 0,Y 537.546,Z 631.852,A -85,B 0,C 180,E1 -3872.997,E2 -3872.997} C_VEL
LIN {X 0,Y 537.577,Z 630.436,A -85,B 0,C 180,E1 -3873.747,E2 -3873.747} C_VEL
LIN {X 0,Y 537.578,Z 626.304,A -85,B 0,C 180,E1 -3875.25,E2 -3875.25} C_VEL
LIN {X 0,Y 537.601,Z 622.616,A -85,B 0,C 180,E1 -3876.29,E2 -3876.29} C_VEL
LIN {X 0,Y 537.698,Z 617.226,A -85,B 0,C 180,E1 -3877.509,E2 -3877.509} C_VEL
LIN {X 0,Y 537.824,Z 611.13,A -85,B 0,C 180,E1 -3878.642,E2 -3878.642} C_VEL
LIN {X 0,Y 537.94,Z 605.139,A -85,B 0,C 180,E1 -3879.588,E2 -3879.588} C_VEL
LIN {X 0,Y 538.119,Z 598.154,A -85,B 0,C 180,E1 -3880.534,E2 -3880.534} C_VEL
LIN {X 0,Y 538.324,Z 590.418,A -85,B 0,C 180,E1 -3881.436,E2 -3881.436} C_VEL
LIN {X 0,Y 538.535,Z 581.361,A -85,B 0,C 180,E1 -3882.338,E2 -3882.338} C_VEL
LIN {X 0,Y 538.775,Z 572.43,A -85,B 0,C 180,E1 -3883.099,E2 -3883.099} C_VEL
LIN {X 0,Y 539.033,Z 563.296,A -85,B 0,C 180,E1 -3883.764,E2 -3883.764} C_VEL
LIN {X 0,Y 539.321,Z 552.371,A -85,B 0,C 180,E1 -3884.43,E2 -3884.43} C_VEL
LIN {X 0,Y 539.568,Z 540.88,A -85,B 0,C 180,E1 -3885.002,E2 -3885.002} C_VEL
LIN {X 0,Y 539.807,Z 529.942,A -85,B 0,C 180,E1 -3885.433,E2 -3885.433} C_VEL
LIN {X 0,Y 539.984,Z 517.822,A -85,B 0,C 180,E1 -3885.796,E2 -3885.796} C_VEL
LIN {X 0,Y 540.166,Z 503.972,A -85,B 0,C 180,E1 -3886.073,E2 -3886.073} C_VEL
LIN {X 0,Y 540.668,Z 382.927,A -85,B 0,C 180,E1 -3887.707,E2 -3887.707} C_VEL
LIN {X 0,Y 538.805,Z 372.469,A -85,B 0,C 180,E1 -3887.93,E2 -3887.93} C_VEL
LIN {X 0,Y 538.834,Z 370.01,A -85,B 0,C 180,E1 -3888.241,E2 -3888.241} C_VEL
LIN {X 0,Y 539.231,Z 351.698,A -85,B 0,C 180,E1 -3891.002,E2 -3891.002} C_VEL
LIN {X 0,Y 539.544,Z 339.905,A -85,B 0,C 180,E1 -3892.802,E2 -3892.802} C_VEL
LIN {X 0,Y 538.061,Z 332.317,A -85,B 0,C 180,E1 -3894.068,E2 -3894.068} C_VEL
LIN {X 0,Y 538.048,Z 332.081,A -85,B 0,C 180,E1 -3895.673,E2 -3895.673} C_VEL
LIN {X 0,Y 538.047,Z 332.088,A -85,B 0,C 180,E1 -3898.048,E2 -3898.048} C_VEL
LIN {X 0,Y 538.026,Z 332.09,A -85,B 0,C 180,E1 -3900.625,E2 -3900.625} C_VEL
LIN {X 0,Y 538.041,Z 332.084,A -85,B 0,C 180,E1 -3903.282,E2 -3903.282} C_VEL
LIN {X 0,Y 538.024,Z 332.091,A -85,B 0,C 180,E1 -3906.001,E2 -3906.001} C_VEL
LIN {X 0,Y 538.012,Z 332.087,A -85,B 0,C 180,E1 -3908.829,E2 -3908.829} C_VEL
LIN {X 0,Y 538.073,Z 332.079,A -85,B 0,C 180,E1 -3910.772,E2 -3910.772} C_VEL
LIN {X 0,Y 538.023,Z 332.088,A -85,B 0,C 180,E1 -3914.074,E2 -3914.074} C_VEL
LIN {X 0,Y 538.019,Z 332.087,A -85,B 0,C 180,E1 -3917.214,E2 -3917.214} C_VEL
LIN {X 0,Y 538.048,Z 332.083,A -85,B 0,C 180,E1 -3920.205,E2 -3920.205} C_VEL
LIN {X 0,Y 538.021,Z 332.08,A -85,B 0,C 180,E1 -3923.067,E2 -3923.067} C_VEL
LIN {X 0,Y 538.024,Z 332.094,A -85,B 0,C 180,E1 -3925.827,E2 -3925.827} C_VEL
LIN {X 0,Y 538.016,Z 332.085,A -85,B 0,C 180,E1 -3928.499,E2 -3928.499} C_VEL
LIN {X 0,Y 538.05,Z 332.074,A -85,B 0,C 180,E1 -3931.099,E2 -3931.099} C_VEL
LIN {X 0,Y 538.042,Z 332.089,A -85,B 0,C 180,E1 -3933.633,E2 -3933.633} C_VEL
LIN {X 0,Y 538.032,Z 332.087,A -85,B 0,C 180,E1 -3936.113,E2 -3936.113} C_VEL
LIN {X 0,Y 538.034,Z 332.089,A -85,B 0,C 180,E1 -3939.348,E2 -3939.348} C_VEL
LIN {X 0,Y 538.062,Z 332.081,A -85,B 0,C 180,E1 -3942.517,E2 -3942.517} C_VEL
LIN {X 0,Y 538.054,Z 332.086,A -85,B 0,C 180,E1 -3945.63,E2 -3945.63} C_VEL
LIN {X 0,Y 538.089,Z 332.079,A -85,B 0,C 180,E1 -3948.702,E2 -3948.702} C_VEL
LIN {X 0,Y 538.083,Z 332.079,A -85,B 0,C 180,E1 -3951.739,E2 -3951.739} C_VEL
LIN {X 0,Y 538.177,Z 332.071,A -85,B 0,C 180,E1 -3954.755,E2 -3954.755} C_VEL
LIN {X 0,Y 538.159,Z 332.069,A -85,B 0,C 180,E1 -3957.755,E2 -3957.755} C_VEL
LIN {X 0,Y 538.179,Z 332.073,A -85,B 0,C 180,E1 -3960.748,E2 -3960.748} C_VEL
LIN {X 0,Y 538.136,Z 332.076,A -85,B 0,C 180,E1 -3962.994,E2 -3962.994} C_VEL
LIN {X 0,Y 538.116,Z 332.074,A -85,B 0,C 180,E1 -3965.997,E2 -3965.997} C_VEL
LIN {X 0,Y 538.069,Z 332.082,A -85,B 0,C 180,E1 -3969.018,E2 -3969.018} C_VEL
LIN {X 0,Y 538.074,Z 332.08,A -85,B 0,C 180,E1 -3972.063,E2 -3972.063} C_VEL
LIN {X 0,Y 538.036,Z 332.083,A -85,B 0,C 180,E1 -3975.144,E2 -3975.144} C_VEL
LIN {X 0,Y 538.027,Z 332.089,A -85,B 0,C 180,E1 -3978.27,E2 -3978.27} C_VEL
LIN {X 0,Y 538.033,Z 332.09,A -85,B 0,C 180,E1 -3980.652,E2 -3980.652} C_VEL
LIN {X 0,Y 538.031,Z 332.086,A -85,B 0,C 180,E1 -3983.887,E2 -3983.887} C_VEL
LIN {X 0,Y 538.041,Z 332.09,A -85,B 0,C 180,E1 -3986.367,E2 -3986.367} C_VEL
LIN {X 0,Y 538.023,Z 332.077,A -85,B 0,C 180,E1 -3988.935,E2 -3988.935} C_VEL
LIN {X 0,Y 538.019,Z 332.086,A -85,B 0,C 180,E1 -3991.891,E2 -3991.891} C_VEL
LIN {X 0,Y 538.025,Z 332.09,A -85,B 0,C 180,E1 -3994.622,E2 -3994.622} C_VEL
LIN {X 0,Y 537.999,Z 332.081,A -85,B 0,C 180,E1 -3997.171,E2 -3997.171} C_VEL
LIN {X 0,Y 538.047,Z 332.082,A -85,B 0,C 180,E1 -3999.795,E2 -3999.795} C_VEL
LIN {X 0,Y 538.018,Z 332.087,A -85,B 0,C 180,E1 -4002.786,E2 -4002.786} C_VEL
LIN {X 0,Y 538.022,Z 332.087,A -85,B 0,C 180,E1 -4005.926,E2 -4005.926} C_VEL
LIN {X 0,Y 538.072,Z 332.079,A -85,B 0,C 180,E1 -4009.25,E2 -4009.25} C_VEL
LIN {X 0,Y 537.99,Z 332.099,A -85,B 0,C 180,E1 -4012.124,E2 -4012.124} C_VEL
LIN {X 0,Y 538.018,Z 332.087,A -85,B 0,C 180,E1 -4014.919,E2 -4014.919} C_VEL
LIN {X 0,Y 538.029,Z 332.089,A -85,B 0,C 180,E1 -4017.619,E2 -4017.619} C_VEL
LIN {X 0,Y 538.04,Z 332.079,A -85,B 0,C 180,E1 -4020.242,E2 -4020.242} C_VEL
LIN {X 0,Y 538.069,Z 332.084,A -85,B 0,C 180,E1 -4022.798,E2 -4022.798} C_VEL
LIN {X 0,Y 538.029,Z 332.093,A -85,B 0,C 180,E1 -4025.705,E2 -4025.705} C_VEL
LIN {X 0,Y 538.053,Z 332.321,A -85,B 0,C 180,E1 -4025.977,E2 -4025.977} C_VEL
LIN {X 0,Y 539.505,Z 339.601,A -85,B 0,C 180,E1 -4027.194,E2 -4027.194} C_VEL
LIN {X 0,Y 539.113,Z 357.597,A -85,B 0,C 180,E1 -4029.938,E2 -4029.938} C_VEL
LIN {X 0,Y 538.782,Z 372.071,A -85,B 0,C 180,E1 -4032.087,E2 -4032.087} C_VEL
LIN {X 0,Y 539.602,Z 376.553,A -85,B 0,C 180,E1 -4032.215,E2 -4032.215} C_VEL
LIN {X 0,Y 540.648,Z 382.852,A -85,B 0,C 180,E1 -4032.336,E2 -4032.336} C_VEL
LIN {X 0,Y 540.103,Z 508.696,A -85,B 0,C 180,E1 -4034.046,E2 -4034.046} C_VEL
LIN {X 0,Y 539.923,Z 523.279,A -85,B 0,C 180,E1 -4034.392,E2 -4034.392} C_VEL
LIN {X 0,Y 539.663,Z 537.719,A -85,B 0,C 180,E1 -4034.904,E2 -4034.904} C_VEL
LIN {X 0,Y 539.398,Z 549.89,A -85,B 0,C 180,E1 -4035.475,E2 -4035.475} C_VEL
LIN {X 0,Y 539.053,Z 562.69,A -85,B 0,C 180,E1 -4036.236,E2 -4036.236} C_VEL
LIN {X 0,Y 538.737,Z 574.318,A -85,B 0,C 180,E1 -4037.092,E2 -4037.092} C_VEL
LIN {X 0,Y 538.454,Z 585.426,A -85,B 0,C 180,E1 -4038.087,E2 -4038.087} C_VEL
LIN {X 0,Y 538.228,Z 594.715,A -85,B 0,C 180,E1 -4039.087,E2 -4039.087} C_VEL
LIN {X 0,Y 537.976,Z 603.563,A -85,B 0,C 180,E1 -4040.223,E2 -4040.223} C_VEL
LIN {X 0,Y 537.823,Z 612.04,A -85,B 0,C 180,E1 -4041.547,E2 -4041.547} C_VEL
LIN {X 0,Y 537.66,Z 618.867,A -85,B 0,C 180,E1 -4042.868,E2 -4042.868} C_VEL
LIN {X 0,Y 537.654,Z 624.963,A -85,B 0,C 180,E1 -4044.375,E2 -4044.375} C_VEL
LIN {X 0,Y 537.55,Z 628.449,A -85,B 0,C 180,E1 -4045.502,E2 -4045.502} C_VEL
LIN {X 0,Y 537.547,Z 631.838,A -85,B 0,C 180,E1 -4047.003,E2 -4047.003} C_VEL
LIN {X 0,Y 537.447,Z 633.837,A -85,B 0,C 180,E1 -4048.502,E2 -4048.502} C_VEL
LIN {X 0,Y 537.44,Z 634.5,A -85,B 0,C 180,E1 -4050.001,E2 -4050.001} C_VEL
LIN {X 0,Y 537.447,Z 633.834,A -85,B 0,C 180,E1 -4051.5,E2 -4051.5} C_VEL
LIN {X 0,Y 537.547,Z 631.831,A -85,B 0,C 180,E1 -4052.999,E2 -4052.999} C_VEL
LIN {X 0,Y 537.55,Z 628.441,A -85,B 0,C 180,E1 -4054.5,E2 -4054.5} C_VEL
LIN {X 0,Y 537.648,Z 623.565,A -85,B 0,C 180,E1 -4056.004,E2 -4056.004} C_VEL
LIN {X 0,Y 537.705,Z 617.05,A -85,B 0,C 180,E1 -4057.511,E2 -4057.511} C_VEL
LIN {X 0,Y 537.86,Z 609.797,A -85,B 0,C 180,E1 -4058.833,E2 -4058.833} C_VEL
LIN {X 0,Y 538.049,Z 600.815,A -85,B 0,C 180,E1 -4060.157,E2 -4060.157} C_VEL
LIN {X 0,Y 538.32,Z 591.383,A -85,B 0,C 180,E1 -4061.294,E2 -4061.294} C_VEL
LIN {X 0,Y 538.566,Z 580.942,A -85,B 0,C 180,E1 -4062.339,E2 -4062.339} C_VEL
LIN {X 0,Y 538.872,Z 569.413,A -85,B 0,C 180,E1 -4063.29,E2 -4063.29} C_VEL
LIN {X 0,Y 539.233,Z 556.62,A -85,B 0,C 180,E1 -4064.146,E2 -4064.146} C_VEL
LIN {X 0,Y 539.518,Z 544.132,A -85,B 0,C 180,E1 -4064.813,E2 -4064.813} C_VEL
LIN {X 0,Y 539.824,Z 531.002,A -85,B 0,C 180,E1 -4065.355,E2 -4065.355} C_VEL
LIN {X 0,Y 540.011,Z 517.401,A -85,B 0,C 180,E1 -4065.766,E2 -4065.766} C_VEL
LIN {X 0,Y 540.146,Z 502.544,A -85,B 0,C 180,E1 -4066.052,E2 -4066.052} C_VEL
LIN {X 0,Y 540.65,Z 382.054,A -85,B 0,C 180,E1 -4067.675,E2 -4067.675} C_VEL
LIN {X 0,Y 538.805,Z 372.262,A -85,B 0,C 180,E1 -4067.898,E2 -4067.898} C_VEL
LIN {X 0,Y 539.157,Z 355.806,A -85,B 0,C 180,E1 -4070.333,E2 -4070.333} C_VEL
LIN {X 0,Y 539.51,Z 339.597,A -85,B 0,C 180,E1 -4072.806,E2 -4072.806} C_VEL
LIN {X 0,Y 538.037,Z 332.173,A -85,B 0,C 180,E1 -4074.072,E2 -4074.072} C_VEL
LIN {X 0,Y 538.047,Z 332.088,A -85,B 0,C 180,E1 -4076.367,E2 -4076.367} C_VEL
LIN {X 0,Y 538.036,Z 332.081,A -85,B 0,C 180,E1 -4078.934,E2 -4078.934} C_VEL
LIN {X 0,Y 538.015,Z 332.095,A -85,B 0,C 180,E1 -4081.888,E2 -4081.888} C_VEL
LIN {X 0,Y 538.037,Z 332.088,A -85,B 0,C 180,E1 -4084.621,E2 -4084.621} C_VEL
LIN {X 0,Y 538.013,Z 332.09,A -85,B 0,C 180,E1 -4087.171,E2 -4087.171} C_VEL
LIN {X 0,Y 538.028,Z 332.093,A -85,B 0,C 180,E1 -4089.797,E2 -4089.797} C_VEL
LIN {X 0,Y 538.023,Z 332.087,A -85,B 0,C 180,E1 -4092.786,E2 -4092.786} C_VEL
LIN {X 0,Y 538.035,Z 332.093,A -85,B 0,C 180,E1 -4095.926,E2 -4095.926} C_VEL
LIN {X 0,Y 538.053,Z 332.086,A -85,B 0,C 180,E1 -4099.253,E2 -4099.253} C_VEL
LIN {X 0,Y 537.996,Z 332.095,A -85,B 0,C 180,E1 -4102.123,E2 -4102.123} C_VEL
LIN {X 0,Y 538.002,Z 332.091,A -85,B 0,C 180,E1 -4104.916,E2 -4104.916} C_VEL
LIN {X 0,Y 538.023,Z 332.096,A -85,B 0,C 180,E1 -4107.618,E2 -4107.618} C_VEL
LIN {X 0,Y 538.021,Z 332.091,A -85,B 0,C 180,E1 -4110.239,E2 -4110.239} C_VEL
LIN {X 0,Y 538.068,Z 332.086,A -85,B 0,C 180,E1 -4112.796,E2 -4112.796} C_VEL
LIN {X 0,Y 538.097,Z 332.312,A -85,B 0,C 180,E1 -4114.014,E2 -4114.014} C_VEL
LIN {X 0,Y 539.547,Z 341.037,A -85,B 0,C 180,E1 -4115.16,E2 -4115.16} C_VEL
LIN {X 0,Y 539.377,Z 360.697,A -85,B 0,C 180,E1 -4117.617,E2 -4117.617} C_VEL
LIN {X 0,Y 539.122,Z 381.351,A -85,B 0,C 180,E1 -4120.188,E2 -4120.188} C_VEL
LIN {X 0,Y 538.805,Z 401.186,A -85,B 0,C 180,E1 -4122.738,E2 -4122.738} C_VEL
LIN {X 0,Y 538.538,Z 420.929,A -85,B 0,C 180,E1 -4125.246,E2 -4125.246} C_VEL
LIN {X 0,Y 538.829,Z 423.231,A -85,B 0,C 180,E1 -4125.326,E2 -4125.326} C_VEL
LIN {X 0,Y 539.67,Z 430.699,A -85,B 0,C 180,E1 -4125.456,E2 -4125.456} C_VEL
LIN {X 0,Y 539.303,Z 529.619,A -85,B 0,C 180,E1 -4126.794,E2 -4126.794} C_VEL
LIN {X 0,Y 539.168,Z 542.562,A -85,B 0,C 180,E1 -4127.102,E2 -4127.102} C_VEL
LIN {X 0,Y 538.967,Z 554.562,A -85,B 0,C 180,E1 -4127.528,E2 -4127.528} C_VEL
LIN {X 0,Y 538.793,Z 566.252,A -85,B 0,C 180,E1 -4128.094,E2 -4128.094} C_VEL
LIN {X 0,Y 538.543,Z 577.689,A -85,B 0,C 180,E1 -4128.807,E2 -4128.807} C_VEL
LIN {X 0,Y 538.306,Z 588.551,A -85,B 0,C 180,E1 -4129.658,E2 -4129.658} C_VEL
LIN {X 0,Y 538.088,Z 598.181,A -85,B 0,C 180,E1 -4130.604,E2 -4130.604} C_VEL
LIN {X 0,Y 537.898,Z 607.527,A -85,B 0,C 180,E1 -4131.737,E2 -4131.737} C_VEL
LIN {X 0,Y 537.745,Z 614.975,A -85,B 0,C 180,E1 -4132.868,E2 -4132.868} C_VEL
LIN {X 0,Y 537.695,Z 620.961,A -85,B 0,C 180,E1 -4133.998,E2 -4133.998} C_VEL
LIN {X 0,Y 537.54,Z 625.699,A -85,B 0,C 180,E1 -4135.125,E2 -4135.125} C_VEL
LIN {X 0,Y 537.592,Z 629.328,A -85,B 0,C 180,E1 -4136.252,E2 -4136.252} C_VEL
LIN {X 0,Y 537.552,Z 631.197,A -85,B 0,C 180,E1 -4137.002,E2 -4137.002} C_VEL
LIN {X 0,Y 537.489,Z 632.631,A -85,B 0,C 180,E1 -4137.752,E2 -4137.752} C_VEL
LIN {X 0,Y 537.442,Z 634.256,A -85,B 0,C 180,E1 -4139.251,E2 -4139.251} C_VEL
LIN {X 0,Y 537.442,Z 634.496,A -85,B 0,C 180,E1 -4140,E2 -4140} C_VEL
LIN {X 0,Y 537.442,Z 634.313,A -85,B 0,C 180,E1 -4140.749,E2 -4140.749} C_VEL
LIN {X 0,Y 537.489,Z 632.764,A -85,B 0,C 180,E1 -4142.248,E2 -4142.248} C_VEL
LIN {X 0,Y 537.552,Z 631.403,A -85,B 0,C 180,E1 -4142.998,E2 -4142.998} C_VEL
LIN {X 0,Y 537.604,Z 628.532,A -85,B 0,C 180,E1 -4144.123,E2 -4144.123} C_VEL
LIN {X 0,Y 537.587,Z 624.633,A -85,B 0,C 180,E1 -4145.251,E2 -4145.251} C_VEL
LIN {X 0,Y 537.68,Z 618.509,A -85,B 0,C 180,E1 -4146.586,E2 -4146.586} C_VEL
LIN {X 0,Y 537.818,Z 612.034,A -85,B 0,C 180,E1 -4147.698,E2 -4147.698} C_VEL
LIN {X 0,Y 537.957,Z 603.859,A -85,B 0,C 180,E1 -4148.83,E2 -4148.83} C_VEL
